LIN {X 0,Y 200.12,Z 814.334,A -85,B 0,C 180,E1 -21665.076,E2 -21665.076} C_VEL
LIN {X 0,Y 196.746,Z 821.173,A -85,B 0,C 180,E1 -21668.43,E2 -21668.43} C_VEL
LIN {X 0,Y 193.868,Z 826.716,A -85,B 0,C 180,E1 -21672.053,E2 -21672.053} C_VEL
LIN {X 0,Y 192.13,Z 830.236,A -85,B 0,C 180,E1 -21675.164,E2 -21675.164} C_VEL
LIN {X 0,Y 190.908,Z 833.5,A -85,B 0,C 180,E1 -21679.394,E2 -21679.394} C_VEL
LIN {X 0,Y 190.669,Z 835.111,A -85,B 0,C 180,E1 -21683.651,E2 -21683.651} C_VEL
LIN {X 0,Y 190.811,Z 835.331,A -85,B 0,C 180,E1 -21685.776,E2 -21685.776} C_VEL
LIN {X 0,Y 191.054,Z 835.155,A -85,B 0,C 180,E1 -21687.892,E2 -21687.892} C_VEL
LIN {X 0,Y 191.378,Z 834.552,A -85,B 0,C 180,E1 -21690,E2 -21690} C_VEL
LIN {X 0,Y 191.229,Z 834.099,A -85,B 0,C 180,E1 -21691.316,E2 -21691.316} C_VEL
LIN {X 0,Y 190.842,Z 834.419,A -85,B 0,C 180,E1 -21694.224,E2 -21694.224} C_VEL
LIN {X 0,Y 190.669,Z 834.183,A -85,B 0,C 180,E1 -21696.349,E2 -21696.349} C_VEL
LIN {X 0,Y 190.908,Z 832.465,A -85,B 0,C 180,E1 -21700.607,E2 -21700.607} C_VEL
LIN {X 0,Y 191.406,Z 831.027,A -85,B 0,C 180,E1 -21702.727,E2 -21702.727} C_VEL
LIN {X 0,Y 192.699,Z 828.062,A -85,B 0,C 180,E1 -21705.874,E2 -21705.874} C_VEL
LIN {X 0,Y 194.57,Z 824.088,A -85,B 0,C 180,E1 -21708.97,E2 -21708.97} C_VEL
LIN {X 0,Y 197.251,Z 818.323,A -85,B 0,C 180,E1 -21712.357,E2 -21712.357} C_VEL
LIN {X 0,Y 200.567,Z 811.407,A -85,B 0,C 180,E1 -21715.419,E2 -21715.419} C_VEL
LIN {X 0,Y 204.393,Z 803.243,A -85,B 0,C 180,E1 -21718.215,E2 -21718.215} C_VEL
LIN {X 0,Y 208.013,Z 794.924,A -85,B 0,C 180,E1 -21720.45,E2 -21720.45} C_VEL
LIN {X 0,Y 211.981,Z 784.694,A -85,B 0,C 180,E1 -21722.598,E2 -21722.598} C_VEL
LIN {X 0,Y 215.942,Z 773.194,A -85,B 0,C 180,E1 -21724.435,E2 -21724.435} C_VEL
LIN {X 0,Y 219.213,Z 761.827,A -85,B 0,C 180,E1 -21725.809,E2 -21725.809} C_VEL
LIN {X 0,Y 222.141,Z 748.843,A -85,B 0,C 180,E1 -21726.949,E2 -21726.949} C_VEL
LIN {X 0,Y 224.167,Z 736.06,A -85,B 0,C 180,E1 -21727.741,E2 -21727.741} C_VEL
LIN {X 0,Y 225.387,Z 722.837,A -85,B 0,C 180,E1 -21728.242,E2 -21728.242} C_VEL
LIN {X 0,Y 227.028,Z 691.593,A -85,B 0,C 180,E1 -21729.201,E2 -21729.201} C_VEL
LIN {X 0,Y 225.581,Z 668.952,A -85,B 0,C 180,E1 -21730.555,E2 -21730.555} C_VEL
LIN {X 0,Y 224.9,Z 662.654,A -85,B 0,C 180,E1 -21731.012,E2 -21731.012} C_VEL
LIN {X 0,Y 219.226,Z 646.641,A -85,B 0,C 180,E1 -21733.317,E2 -21733.317} C_VEL
LIN {X 0,Y 217.376,Z 642.169,A -85,B 0,C 180,E1 -21734.081,E2 -21734.081} C_VEL
LIN {X 0,Y 210.802,Z 631.796,A -85,B 0,C 180,E1 -21736.717,E2 -21736.717} C_VEL
LIN {X 0,Y 205.693,Z 624.408,A -85,B 0,C 180,E1 -21738.968,E2 -21738.968} C_VEL
LIN {X 0,Y 202.878,Z 620.482,A -85,B 0,C 180,E1 -21740.305,E2 -21740.305} C_VEL
LIN {X 0,Y 200.044,Z 616.68,A -85,B 0,C 180,E1 -21741.734,E2 -21741.734} C_VEL
LIN {X 0,Y 197.692,Z 613.872,A -85,B 0,C 180,E1 -21742.973,E2 -21742.973} C_VEL
LIN {X 0,Y 196.534,Z 611.954,A -85,B 0,C 180,E1 -21743.647,E2 -21743.647} C_VEL
LIN {X 0,Y 194.085,Z 610.022,A -85,B 0,C 180,E1 -21744.99,E2 -21744.99} C_VEL
LIN {X 0,Y 192.896,Z 607.766,A -85,B 0,C 180,E1 -21745.774,E2 -21745.774} C_VEL
LIN {X 0,Y 192.586,Z 606.475,A -85,B 0,C 180,E1 -21746.106,E2 -21746.106} C_VEL
LIN {X 0,Y 192.657,Z 606.463,A -85,B 0,C 180,E1 -21751.691,E2 -21751.691} C_VEL
LIN {X 0,Y 192.702,Z 606.457,A -85,B 0,C 180,E1 -21756.348,E2 -21756.348} C_VEL
LIN {X 0,Y 192.778,Z 606.466,A -85,B 0,C 180,E1 -21761.414,E2 -21761.414} C_VEL
LIN {X 0,Y 192.757,Z 606.449,A -85,B 0,C 180,E1 -21765.213,E2 -21765.213} C_VEL
LIN {X 0,Y 192.941,Z 606.428,A -85,B 0,C 180,E1 -21769.566,E2 -21769.566} C_VEL
LIN {X 0,Y 192.982,Z 606.438,A -85,B 0,C 180,E1 -21773.728,E2 -21773.728} C_VEL
LIN {X 0,Y 193.259,Z 606.38,A -85,B 0,C 180,E1 -21777.916,E2 -21777.916} C_VEL
LIN {X 0,Y 193.439,Z 606.366,A -85,B 0,C 180,E1 -21780,E2 -21780} C_VEL
LIN {X 0,Y 192.973,Z 606.424,A -85,B 0,C 180,E1 -21784.177,E2 -21784.177} C_VEL
LIN {X 0,Y 193.057,Z 606.432,A -85,B 0,C 180,E1 -21788.373,E2 -21788.373} C_VEL
LIN {X 0,Y 192.805,Z 606.44,A -85,B 0,C 180,E1 -21792.633,E2 -21792.633} C_VEL
LIN {X 0,Y 192.754,Z 606.463,A -85,B 0,C 180,E1 -21796.959,E2 -21796.959} C_VEL
LIN {X 0,Y 192.7,Z 606.473,A -85,B 0,C 180,E1 -21802.8,E2 -21802.8} C_VEL
LIN {X 0,Y 192.73,Z 606.629,A -85,B 0,C 180,E1 -21803.008,E2 -21803.008} C_VEL
LIN {X 0,Y 193.555,Z 609.094,A -85,B 0,C 180,E1 -21803.628,E2 -21803.628} C_VEL
LIN {X 0,Y 195.51,Z 611.341,A -85,B 0,C 180,E1 -21804.775,E2 -21804.775} C_VEL
LIN {X 0,Y 196.99,Z 612.434,A -85,B 0,C 180,E1 -21805.561,E2 -21805.561} C_VEL
LIN {X 0,Y 198.774,Z 615.45,A -85,B 0,C 180,E1 -21806.582,E2 -21806.582} C_VEL
LIN {X 0,Y 200.997,Z 617.62,A -85,B 0,C 180,E1 -21807.693,E2 -21807.693} C_VEL
LIN {X 0,Y 203.451,Z 621.161,A -85,B 0,C 180,E1 -21808.922,E2 -21808.922} C_VEL
LIN {X 0,Y 204.958,Z 622.964,A -85,B 0,C 180,E1 -21809.621,E2 -21809.621} C_VEL
LIN {X 0,Y 208.923,Z 628.481,A -85,B 0,C 180,E1 -21811.403,E2 -21811.403} C_VEL
LIN {X 0,Y 211.895,Z 632.606,A -85,B 0,C 180,E1 -21812.651,E2 -21812.651} C_VEL
LIN {X 0,Y 216.538,Z 639.553,A -85,B 0,C 180,E1 -21814.492,E2 -21814.492} C_VEL
LIN {X 0,Y 222.348,Z 649.031,A -85,B 0,C 180,E1 -21816.633,E2 -21816.633} C_VEL
LIN {X 0,Y 228.602,Z 660.543,A -85,B 0,C 180,E1 -21818.785,E2 -21818.785} C_VEL
LIN {X 0,Y 229.105,Z 661.475,A -85,B 0,C 180,E1 -21818.949,E2 -21818.949} C_VEL
LIN {X 0,Y 227.497,Z 690.233,A -85,B 0,C 180,E1 -21819.801,E2 -21819.801} C_VEL
LIN {X 0,Y 226.656,Z 704.192,A -85,B 0,C 180,E1 -21820.346,E2 -21820.346} C_VEL
LIN {X 0,Y 225.1,Z 717.435,A -85,B 0,C 180,E1 -21821.184,E2 -21821.184} C_VEL
LIN {X 0,Y 223.055,Z 729.09,A -85,B 0,C 180,E1 -21822.233,E2 -21822.233} C_VEL
LIN {X 0,Y 220.152,Z 741.552,A -85,B 0,C 180,E1 -21823.76,E2 -21823.76} C_VEL
LIN {X 0,Y 217.15,Z 751.905,A -85,B 0,C 180,E1 -21825.4,E2 -21825.4} C_VEL
LIN {X 0,Y 213.801,Z 761.515,A -85,B 0,C 180,E1 -21827.315,E2 -21827.315} C_VEL
LIN {X 0,Y 210.529,Z 769.77,A -85,B 0,C 180,E1 -21829.387,E2 -21829.387} C_VEL
LIN {X 0,Y 206.528,Z 778.67,A -85,B 0,C 180,E1 -21832.229,E2 -21832.229} C_VEL
LIN {X 0,Y 203.016,Z 785.739,A -85,B 0,C 180,E1 -21835.167,E2 -21835.167} C_VEL
LIN {X 0,Y 199.876,Z 791.284,A -85,B 0,C 180,E1 -21838.169,E2 -21838.169} C_VEL
LIN {X 0,Y 197.26,Z 795.562,A -85,B 0,C 180,E1 -21841.251,E2 -21841.251} C_VEL
LIN {X 0,Y 195.123,Z 798.71,A -85,B 0,C 180,E1 -21844.392,E2 -21844.392} C_VEL
LIN {X 0,Y 193.95,Z 800.243,A -85,B 0,C 180,E1 -21846.51,E2 -21846.51} C_VEL
LIN {X 0,Y 193.004,Z 801.338,A -85,B 0,C 180,E1 -21848.646,E2 -21848.646} C_VEL
LIN {X 0,Y 191.694,Z 802.23,A -85,B 0,C 180,E1 -21852.945,E2 -21852.945} C_VEL
LIN {X 0,Y 191.283,Z 802.087,A -85,B 0,C 180,E1 -21855.097,E2 -21855.097} C_VEL
LIN {X 0,Y 191.049,Z 801.498,A -85,B 0,C 180,E1 -21857.249,E2 -21857.249} C_VEL
LIN {X 0,Y 191.12,Z 799.132,A -85,B 0,C 180,E1 -21861.542,E2 -21861.542} C_VEL
LIN {X 0,Y 191.571,Z 796.233,A -85,B 0,C 180,E1 -21864.738,E2 -21864.738} C_VEL
LIN {X 0,Y 192.37,Z 792.307,A -85,B 0,C 180,E1 -21867.906,E2 -21867.906} C_VEL
LIN {X 0,Y 193.447,Z 787.253,A -85,B 0,C 180,E1 -21871.041,E2 -21871.041} C_VEL
LIN {X 0,Y 194.896,Z 780.879,A -85,B 0,C 180,E1 -21874.136,E2 -21874.136} C_VEL
LIN {X 0,Y 196.846,Z 772.934,A -85,B 0,C 180,E1 -21877.178,E2 -21877.178} C_VEL
LIN {X 0,Y 198.856,Z 764.808,A -85,B 0,C 180,E1 -21879.664,E2 -21879.664} C_VEL
LIN {X 0,Y 200.966,Z 754.894,A -85,B 0,C 180,E1 -21882.112,E2 -21882.112} C_VEL
LIN {X 0,Y 203.25,Z 743.364,A -85,B 0,C 180,E1 -21884.328,E2 -21884.328} C_VEL
LIN {X 0,Y 204.991,Z 732.793,A -85,B 0,C 180,E1 -21885.918,E2 -21885.918} C_VEL
LIN {X 0,Y 206.257,Z 723.793,A -85,B 0,C 180,E1 -21886.978,E2 -21886.978} C_VEL
LIN {X 0,Y 206.049,Z 721.845,A -85,B 0,C 180,E1 -21887.246,E2 -21887.246} C_VEL
LIN {X 0,Y 205.46,Z 720.362,A -85,B 0,C 180,E1 -21887.495,E2 -21887.495} C_VEL
LIN {X 0,Y 203.842,Z 732.893,A -85,B 0,C 180,E1 -21888.988,E2 -21888.988} C_VEL
LIN {X 0,Y 201.992,Z 744.543,A -85,B 0,C 180,E1 -21890.792,E2 -21890.792} C_VEL
LIN {X 0,Y 200.128,Z 754.446,A -85,B 0,C 180,E1 -21892.723,E2 -21892.723} C_VEL
LIN {X 0,Y 198.076,Z 764.576,A -85,B 0,C 180,E1 -21895.199,E2 -21895.199} C_VEL
LIN {X 0,Y 196.25,Z 773.003,A -85,B 0,C 180,E1 -21897.745,E2 -21897.745} C_VEL
LIN {X 0,Y 194.673,Z 780.071,A -85,B 0,C 180,E1 -21900.359,E2 -21900.359} C_VEL
LIN {X 0,Y 193.143,Z 787.462,A -85,B 0,C 180,E1 -21903.782,E2 -21903.782} C_VEL
LIN {X 0,Y 192.006,Z 793.453,A -85,B 0,C 180,E1 -21907.421,E2 -21907.421} C_VEL
LIN {X 0,Y 191.316,Z 797.226,A -85,B 0,C 180,E1 -21910.425,E2 -21910.425} C_VEL
LIN {X 0,Y 190.912,Z 800.782,A -85,B 0,C 180,E1 -21914.381,E2 -21914.381} C_VEL
LIN {X 0,Y 191.154,Z 802.884,A -85,B 0,C 180,E1 -21918.563,E2 -21918.563} C_VEL
LIN {X 0,Y 191.756,Z 803.442,A -85,B 0,C 180,E1 -21921.46,E2 -21921.46} C_VEL
LIN {X 0,Y 192.666,Z 803.238,A -85,B 0,C 180,E1 -21924.293,E2 -21924.293} C_VEL
LIN {X 0,Y 193.884,Z 802.31,A -85,B 0,C 180,E1 -21927.062,E2 -21927.062} C_VEL
LIN {X 0,Y 196.291,Z 799.661,A -85,B 0,C 180,E1 -21931.095,E2 -21931.095} C_VEL
LIN {X 0,Y 198.467,Z 796.735,A -85,B 0,C 180,E1 -21933.893,E2 -21933.893} C_VEL
LIN {X 0,Y 201.004,Z 792.853,A -85,B 0,C 180,E1 -21936.673,E2 -21936.673} C_VEL
LIN {X 0,Y 204.708,Z 786.776,A -85,B 0,C 180,E1 -21939.921,E2 -21939.921} C_VEL
LIN {X 0,Y 208.621,Z 779.506,A -85,B 0,C 180,E1 -21942.856,E2 -21942.856} C_VEL
LIN {X 0,Y 212.161,Z 772.164,A -85,B 0,C 180,E1 -21945.189,E2 -21945.189} C_VEL
LIN {X 0,Y 216.012,Z 763.265,A -85,B 0,C 180,E1 -21947.43,E2 -21947.43} C_VEL
LIN {X 0,Y 219.818,Z 752.988,A -85,B 0,C 180,E1 -21949.464,E2 -21949.464} C_VEL
LIN {X 0,Y 223.238,Z 741.939,A -85,B 0,C 180,E1 -21951.172,E2 -21951.172} C_VEL
LIN {X 0,Y 226.14,Z 730.481,A -85,B 0,C 180,E1 -21952.556,E2 -21952.556} C_VEL
LIN {X 0,Y 228.608,Z 717.196,A -85,B 0,C 180,E1 -21953.765,E2 -21953.765} C_VEL
LIN {X 0,Y 230.282,Z 704.049,A -85,B 0,C 180,E1 -21954.604,E2 -21954.604} C_VEL
LIN {X 0,Y 233.633,Z 664.942,A -85,B 0,C 180,E1 -21956.045,E2 -21956.045} C_VEL
LIN {X 0,Y 233.694,Z 662.933,A -85,B 0,C 180,E1 -21956.154,E2 -21956.154} C_VEL
LIN {X 0,Y 228.771,Z 653.042,A -85,B 0,C 180,E1 -21958.575,E2 -21958.575} C_VEL
LIN {X 0,Y 223.573,Z 644.616,A -85,B 0,C 180,E1 -21961.401,E2 -21961.401} C_VEL
LIN {X 0,Y 220.882,Z 640.179,A -85,B 0,C 180,E1 -21963.094,E2 -21963.094} C_VEL
LIN {X 0,Y 219.611,Z 638.316,A -85,B 0,C 180,E1 -21963.928,E2 -21963.928} C_VEL
LIN {X 0,Y 216.914,Z 634.667,A -85,B 0,C 180,E1 -21965.899,E2 -21965.899} C_VEL
LIN {X 0,Y 214.346,Z 631.703,A -85,B 0,C 180,E1 -21967.981,E2 -21967.981} C_VEL
LIN {X 0,Y 213.334,Z 629.707,A -85,B 0,C 180,E1 -21969.036,E2 -21969.036} C_VEL
LIN {X 0,Y 210.621,Z 627.078,A -85,B 0,C 180,E1 -21971.915,E2 -21971.915} C_VEL
LIN {X 0,Y 209.368,Z 624.536,A -85,B 0,C 180,E1 -21973.862,E2 -21973.862} C_VEL
LIN {X 0,Y 207.116,Z 623.322,A -85,B 0,C 180,E1 -21978.264,E2 -21978.264} C_VEL
LIN {X 0,Y 206.61,Z 623.792,A -85,B 0,C 180,E1 -21979.887,E2 -21979.887} C_VEL
LIN {X 0,Y 206.124,Z 625.393,A -85,B 0,C 180,E1 -21981.473,E2 -21981.473} C_VEL
LIN {X 0,Y 205.668,Z 631.128,A -85,B 0,C 180,E1 -21985.656,E2 -21985.656} C_VEL
LIN {X 0,Y 205.893,Z 632.049,A -85,B 0,C 180,E1 -21986.744,E2 -21986.744} C_VEL
LIN {X 0,Y 206.917,Z 634.357,A -85,B 0,C 180,E1 -21989.521,E2 -21989.521} C_VEL
LIN {X 0,Y 209.94,Z 639.333,A -85,B 0,C 180,E1 -21994.02,E2 -21994.02} C_VEL
LIN {X 0,Y 213.894,Z 646.761,A -85,B 0,C 180,E1 -21998.085,E2 -21998.085} C_VEL
LIN {X 0,Y 217.081,Z 653.246,A -85,B 0,C 180,E1 -22000.715,E2 -22000.715} C_VEL
LIN {X 0,Y 219.756,Z 658.788,A -85,B 0,C 180,E1 -22002.587,E2 -22002.587} C_VEL
LIN {X 0,Y 223.079,Z 666.597,A -85,B 0,C 180,E1 -22004.746,E2 -22004.746} C_VEL
LIN {X 0,Y 226.39,Z 675.777,A -85,B 0,C 180,E1 -22006.747,E2 -22006.747} C_VEL
LIN {X 0,Y 226.951,Z 691.065,A -85,B 0,C 180,E1 -22008.006,E2 -22008.006} C_VEL
LIN {X 0,Y 226.935,Z 698.487,A -85,B 0,C 180,E1 -22008.49,E2 -22008.49} C_VEL
LIN {X 0,Y 224.042,Z 728.913,A -85,B 0,C 180,E1 -22009.623,E2 -22009.623} C_VEL
LIN {X 0,Y 221.659,Z 742.96,A -85,B 0,C 180,E1 -22010.436,E2 -22010.436} C_VEL
LIN {X 0,Y 218.562,Z 755.539,A -85,B 0,C 180,E1 -22011.464,E2 -22011.464} C_VEL
LIN {X 0,Y 214.895,Z 767.424,A -85,B 0,C 180,E1 -22012.77,E2 -22012.77} C_VEL
LIN {X 0,Y 210.955,Z 778.281,A -85,B 0,C 180,E1 -22014.338,E2 -22014.338} C_VEL
LIN {X 0,Y 206.292,Z 789.283,A -85,B 0,C 180,E1 -22016.386,E2 -22016.386} C_VEL
LIN {X 0,Y 201.372,Z 799.951,A -85,B 0,C 180,E1 -22019.018,E2 -22019.018} C_VEL
LIN {X 0,Y 196.911,Z 808.526,A -85,B 0,C 180,E1 -22021.777,E2 -22021.777} C_VEL
LIN {X 0,Y 192.54,Z 816.583,A -85,B 0,C 180,E1 -22025.181,E2 -22025.181} C_VEL
LIN {X 0,Y 189.62,Z 822.117,A -85,B 0,C 180,E1 -22028.246,E2 -22028.246} C_VEL
LIN {X 0,Y 187.083,Z 826.527,A -85,B 0,C 180,E1 -22031.379,E2 -22031.379} C_VEL
LIN {X 0,Y 185.253,Z 829.916,A -85,B 0,C 180,E1 -22034.6,E2 -22034.6} C_VEL
LIN {X 0,Y 184.403,Z 831.675,A -85,B 0,C 180,E1 -22036.781,E2 -22036.781} C_VEL
LIN {X 0,Y 183.605,Z 833.941,A -85,B 0,C 180,E1 -22041.193,E2 -22041.193} C_VEL
LIN {X 0,Y 183.664,Z 834.63,A -85,B 0,C 180,E1 -22044.215,E2 -22044.215} C_VEL
LIN {X 0,Y 183.971,Z 834.424,A -85,B 0,C 180,E1 -22047.811,E2 -22047.811} C_VEL
LIN {X 0,Y 184.265,Z 833.477,A -85,B 0,C 180,E1 -22050.546,E2 -22050.546} C_VEL
LIN {X 0,Y 183.642,Z 833.713,A -85,B 0,C 180,E1 -22055.717,E2 -22055.717} C_VEL
LIN {X 0,Y 183.603,Z 832.973,A -85,B 0,C 180,E1 -22058.807,E2 -22058.807} C_VEL
LIN {X 0,Y 184.427,Z 830.537,A -85,B 0,C 180,E1 -22063.217,E2 -22063.217} C_VEL
LIN {X 0,Y 185.826,Z 827.63,A -85,B 0,C 180,E1 -22066.478,E2 -22066.478} C_VEL
LIN {X 0,Y 187.843,Z 823.721,A -85,B 0,C 180,E1 -22069.677,E2 -22069.677} C_VEL
LIN {X 0,Y 190.335,Z 818.696,A -85,B 0,C 180,E1 -22072.81,E2 -22072.81} C_VEL
LIN {X 0,Y 193.544,Z 812.421,A -85,B 0,C 180,E1 -22075.832,E2 -22075.832} C_VEL
LIN {X 0,Y 197.446,Z 804.63,A -85,B 0,C 180,E1 -22078.719,E2 -22078.719} C_VEL
LIN {X 0,Y 201.92,Z 794.934,A -85,B 0,C 180,E1 -22081.472,E2 -22081.472} C_VEL
LIN {X 0,Y 206.046,Z 784.901,A -85,B 0,C 180,E1 -22083.659,E2 -22083.659} C_VEL
LIN {X 0,Y 210.153,Z 773.575,A -85,B 0,C 180,E1 -22085.524,E2 -22085.524} C_VEL
LIN {X 0,Y 213.523,Z 762.489,A -85,B 0,C 180,E1 -22086.918,E2 -22086.918} C_VEL
LIN {X 0,Y 216.544,Z 750.025,A -85,B 0,C 180,E1 -22088.071,E2 -22088.071} C_VEL
LIN {X 0,Y 218.826,Z 736.752,A -85,B 0,C 180,E1 -22088.932,E2 -22088.932} C_VEL
LIN {X 0,Y 220.048,Z 725.276,A -85,B 0,C 180,E1 -22089.416,E2 -22089.416} C_VEL
LIN {X 0,Y 221.908,Z 692.411,A -85,B 0,C 180,E1 -22090.44,E2 -22090.44} C_VEL
LIN {X 0,Y 220.639,Z 670.867,A -85,B 0,C 180,E1 -22091.767,E2 -22091.767} C_VEL
LIN {X 0,Y 220.188,Z 665.856,A -85,B 0,C 180,E1 -22092.127,E2 -22092.127} C_VEL
LIN {X 0,Y 215.242,Z 651.377,A -85,B 0,C 180,E1 -22094.268,E2 -22094.268} C_VEL
LIN {X 0,Y 213.378,Z 646.747,A -85,B 0,C 180,E1 -22095.083,E2 -22095.083} C_VEL
LIN {X 0,Y 206.373,Z 635.432,A -85,B 0,C 180,E1 -22098.08,E2 -22098.08} C_VEL
LIN {X 0,Y 200.052,Z 626.343,A -85,B 0,C 180,E1 -22101.111,E2 -22101.111} C_VEL
LIN {X 0,Y 197.181,Z 622.528,A -85,B 0,C 180,E1 -22102.624,E2 -22102.624} C_VEL
LIN {X 0,Y 194.719,Z 619.272,A -85,B 0,C 180,E1 -22104.01,E2 -22104.01} C_VEL
LIN {X 0,Y 194.026,Z 618.292,A -85,B 0,C 180,E1 -22104.422,E2 -22104.422} C_VEL
LIN {X 0,Y 191.421,Z 615.809,A -85,B 0,C 180,E1 -22105.951,E2 -22105.951} C_VEL
LIN {X 0,Y 190.049,Z 613.108,A -85,B 0,C 180,E1 -22106.915,E2 -22106.915} C_VEL
LIN {X 0,Y 187.378,Z 611.316,A -85,B 0,C 180,E1 -22108.64,E2 -22108.64} C_VEL
LIN {X 0,Y 185.921,Z 608.849,A -85,B 0,C 180,E1 -22109.786,E2 -22109.786} C_VEL
LIN {X 0,Y 185.557,Z 607.348,A -85,B 0,C 180,E1 -22110.191,E2 -22110.191} C_VEL
LIN {X 0,Y 185.585,Z 607.353,A -85,B 0,C 180,E1 -22115.382,E2 -22115.382} C_VEL
LIN {X 0,Y 185.691,Z 607.353,A -85,B 0,C 180,E1 -22121.115,E2 -22121.115} C_VEL
LIN {X 0,Y 185.692,Z 607.324,A -85,B 0,C 180,E1 -22124.637,E2 -22124.637} C_VEL
LIN {X 0,Y 185.885,Z 607.308,A -85,B 0,C 180,E1 -22129.418,E2 -22129.418} C_VEL
LIN {X 0,Y 185.945,Z 607.309,A -85,B 0,C 180,E1 -22133.489,E2 -22133.489} C_VEL
LIN {X 0,Y 186.203,Z 607.258,A -85,B 0,C 180,E1 -22137.837,E2 -22137.837} C_VEL
LIN {X 0,Y 186.402,Z 607.241,A -85,B 0,C 180,E1 -22140,E2 -22140} C_VEL
LIN {X 0,Y 185.92,Z 607.3,A -85,B 0,C 180,E1 -22144.336,E2 -22144.336} C_VEL
LIN {X 0,Y 186.004,Z 607.314,A -85,B 0,C 180,E1 -22148.693,E2 -22148.693} C_VEL
LIN {X 0,Y 185.73,Z 607.322,A -85,B 0,C 180,E1 -22153.123,E2 -22153.123} C_VEL
LIN {X 0,Y 185.686,Z 607.335,A -85,B 0,C 180,E1 -22157.625,E2 -22157.625} C_VEL
LIN {X 0,Y 185.69,Z 607.389,A -85,B 0,C 180,E1 -22158.884,E2 -22158.884} C_VEL
LIN {X 0,Y 186.351,Z 609.679,A -85,B 0,C 180,E1 -22159.522,E2 -22159.522} C_VEL
LIN {X 0,Y 187.933,Z 611.811,A -85,B 0,C 180,E1 -22160.695,E2 -22160.695} C_VEL
LIN {X 0,Y 190.258,Z 613.373,A -85,B 0,C 180,E1 -22162.177,E2 -22162.177} C_VEL
LIN {X 0,Y 192.032,Z 616.47,A -85,B 0,C 180,E1 -22163.382,E2 -22163.382} C_VEL
LIN {X 0,Y 194.504,Z 618.874,A -85,B 0,C 180,E1 -22164.814,E2 -22164.814} C_VEL
LIN {X 0,Y 196.873,Z 622.256,A -85,B 0,C 180,E1 -22166.172,E2 -22166.172} C_VEL
LIN {X 0,Y 198.553,Z 624.143,A -85,B 0,C 180,E1 -22167.054,E2 -22167.054} C_VEL
LIN {X 0,Y 201.189,Z 627.641,A -85,B 0,C 180,E1 -22168.401,E2 -22168.401} C_VEL
LIN {X 0,Y 205.7,Z 633.976,A -85,B 0,C 180,E1 -22170.543,E2 -22170.543} C_VEL
LIN {X 0,Y 210.561,Z 640.986,A -85,B 0,C 180,E1 -22172.651,E2 -22172.651} C_VEL
LIN {X 0,Y 217.786,Z 652.676,A -85,B 0,C 180,E1 -22175.511,E2 -22175.511} C_VEL
LIN {X 0,Y 223.948,Z 664.331,A -85,B 0,C 180,E1 -22177.767,E2 -22177.767} C_VEL
LIN {X 0,Y 222.381,Z 690.882,A -85,B 0,C 180,E1 -22178.56,E2 -22178.56} C_VEL
LIN {X 0,Y 221.499,Z 704.795,A -85,B 0,C 180,E1 -22179.112,E2 -22179.112} C_VEL
LIN {X 0,Y 219.943,Z 717.573,A -85,B 0,C 180,E1 -22179.926,E2 -22179.926} C_VEL
LIN {X 0,Y 217.734,Z 729.689,A -85,B 0,C 180,E1 -22181.02,E2 -22181.02} C_VEL
LIN {X 0,Y 214.709,Z 742.158,A -85,B 0,C 180,E1 -22182.569,E2 -22182.569} C_VEL
LIN {X 0,Y 211.621,Z 752.417,A -85,B 0,C 180,E1 -22184.22,E2 -22184.22} C_VEL
LIN {X 0,Y 208.093,Z 762.126,A -85,B 0,C 180,E1 -22186.185,E2 -22186.185} C_VEL
LIN {X 0,Y 204.302,Z 771.192,A -85,B 0,C 180,E1 -22188.533,E2 -22188.533} C_VEL
LIN {X 0,Y 200.135,Z 779.954,A -85,B 0,C 180,E1 -22191.443,E2 -22191.443} C_VEL
LIN {X 0,Y 196.45,Z 786.852,A -85,B 0,C 180,E1 -22194.456,E2 -22194.456} C_VEL
LIN {X 0,Y 193.692,Z 791.498,A -85,B 0,C 180,E1 -22197.026,E2 -22197.026} C_VEL
LIN {X 0,Y 190.872,Z 795.87,A -85,B 0,C 180,E1 -22200.194,E2 -22200.194} C_VEL
LIN {X 0,Y 188.581,Z 799.104,A -85,B 0,C 180,E1 -22203.436,E2 -22203.436} C_VEL
LIN {X 0,Y 187.287,Z 800.679,A -85,B 0,C 180,E1 -22205.621,E2 -22205.621} C_VEL
LIN {X 0,Y 186.229,Z 801.838,A -85,B 0,C 180,E1 -22207.829,E2 -22207.829} C_VEL
LIN {X 0,Y 184.87,Z 802.806,A -85,B 0,C 180,E1 -22211.879,E2 -22211.879} C_VEL
LIN {X 0,Y 184.295,Z 802.726,A -85,B 0,C 180,E1 -22214.518,E2 -22214.518} C_VEL
LIN {X 0,Y 184.003,Z 802.211,A -85,B 0,C 180,E1 -22216.752,E2 -22216.752} C_VEL
LIN {X 0,Y 183.917,Z 801.263,A -85,B 0,C 180,E1 -22218.985,E2 -22218.985} C_VEL
LIN {X 0,Y 184.174,Z 798.684,A -85,B 0,C 180,E1 -22222.817,E2 -22222.817} C_VEL
LIN {X 0,Y 184.954,Z 794.679,A -85,B 0,C 180,E1 -22226.733,E2 -22226.733} C_VEL
LIN {X 0,Y 185.89,Z 790.106,A -85,B 0,C 180,E1 -22230,E2 -22230} C_VEL
LIN {X 0,Y 187.555,Z 783.198,A -85,B 0,C 180,E1 -22233.76,E2 -22233.76} C_VEL
LIN {X 0,Y 189.466,Z 775.71,A -85,B 0,C 180,E1 -22236.924,E2 -22236.924} C_VEL
LIN {X 0,Y 191.872,Z 766.274,A -85,B 0,C 180,E1 -22240.019,E2 -22240.019} C_VEL
LIN {X 0,Y 194.054,Z 756.597,A -85,B 0,C 180,E1 -22242.55,E2 -22242.55} C_VEL
LIN {X 0,Y 196.251,Z 745.958,A -85,B 0,C 180,E1 -22244.73,E2 -22244.73} C_VEL
LIN {X 0,Y 198.227,Z 735.059,A -85,B 0,C 180,E1 -22246.477,E2 -22246.477} C_VEL
LIN {X 0,Y 198.855,Z 730.991,A -85,B 0,C 180,E1 -22247.026,E2 -22247.026} C_VEL
LIN {X 0,Y 198.717,Z 729.466,A -85,B 0,C 180,E1 -22247.272,E2 -22247.272} C_VEL
LIN {X 0,Y 197.908,Z 728.01,A -85,B 0,C 180,E1 -22247.638,E2 -22247.638} C_VEL
LIN {X 0,Y 196.084,Z 739.963,A -85,B 0,C 180,E1 -22249.339,E2 -22249.339} C_VEL
LIN {X 0,Y 194.193,Z 750.33,A -85,B 0,C 180,E1 -22251.217,E2 -22251.217} C_VEL
LIN {X 0,Y 191.921,Z 761.382,A -85,B 0,C 180,E1 -22253.753,E2 -22253.753} C_VEL
LIN {X 0,Y 190.008,Z 770.415,A -85,B 0,C 180,E1 -22256.349,E2 -22256.349} C_VEL
LIN {X 0,Y 188.229,Z 778.044,A -85,B 0,C 180,E1 -22259.037,E2 -22259.037} C_VEL
LIN {X 0,Y 186.644,Z 785.381,A -85,B 0,C 180,E1 -22262.27,E2 -22262.27} C_VEL
LIN {X 0,Y 185.317,Z 791.717,A -85,B 0,C 180,E1 -22265.831,E2 -22265.831} C_VEL
LIN {X 0,Y 184.519,Z 795.928,A -85,B 0,C 180,E1 -22268.865,E2 -22268.865} C_VEL
LIN {X 0,Y 184.005,Z 799.206,A -85,B 0,C 180,E1 -22271.918,E2 -22271.918} C_VEL
LIN {X 0,Y 183.824,Z 801.637,A -85,B 0,C 180,E1 -22274.994,E2 -22274.994} C_VEL
LIN {X 0,Y 183.876,Z 802.557,A -85,B 0,C 180,E1 -22276.568,E2 -22276.568} C_VEL
LIN {X 0,Y 184.274,Z 803.743,A -85,B 0,C 180,E1 -22279.708,E2 -22279.708} C_VEL
LIN {X 0,Y 185.093,Z 804.108,A -85,B 0,C 180,E1 -22282.878,E2 -22282.878} C_VEL
LIN {X 0,Y 186.299,Z 803.629,A -85,B 0,C 180,E1 -22286.09,E2 -22286.09} C_VEL
LIN {X 0,Y 187.985,Z 802.249,A -85,B 0,C 180,E1 -22289.3,E2 -22289.3} C_VEL
LIN {X 0,Y 190.144,Z 799.892,A -85,B 0,C 180,E1 -22292.505,E2 -22292.505} C_VEL
LIN {X 0,Y 193.57,Z 795.443,A -85,B 0,C 180,E1 -22296.46,E2 -22296.46} C_VEL
LIN {X 0,Y 197.044,Z 790.349,A -85,B 0,C 180,E1 -22299.65,E2 -22299.65} C_VEL
LIN {X 0,Y 201.205,Z 783.448,A -85,B 0,C 180,E1 -22302.856,E2 -22302.856} C_VEL
LIN {X 0,Y 205.735,Z 774.988,A -85,B 0,C 180,E1 -22305.838,E2 -22305.838} C_VEL
LIN {X 0,Y 210.248,Z 765.258,A -85,B 0,C 180,E1 -22308.43,E2 -22308.43} C_VEL
LIN {X 0,Y 214.364,Z 755.033,A -85,B 0,C 180,E1 -22310.565,E2 -22310.565} C_VEL
LIN {X 0,Y 218.133,Z 743.833,A -85,B 0,C 180,E1 -22312.363,E2 -22312.363} C_VEL
LIN {X 0,Y 221.141,Z 732.709,A -85,B 0,C 180,E1 -22313.763,E2 -22313.763} C_VEL
LIN {X 0,Y 223.738,Z 720.218,A -85,B 0,C 180,E1 -22314.965,E2 -22314.965} C_VEL
LIN {X 0,Y 225.631,Z 706.998,A -85,B 0,C 180,E1 -22315.86,E2 -22315.86} C_VEL
LIN {X 0,Y 226.873,Z 693.522,A -85,B 0,C 180,E1 -22316.448,E2 -22316.448} C_VEL
LIN {X 0,Y 229.279,Z 666.002,A -85,B 0,C 180,E1 -22317.466,E2 -22317.466} C_VEL
LIN {X 0,Y 225.266,Z 657.892,A -85,B 0,C 180,E1 -22319.607,E2 -22319.607} C_VEL
LIN {X 0,Y 219.546,Z 647.958,A -85,B 0,C 180,E1 -22323.07,E2 -22323.07} C_VEL
LIN {X 0,Y 217.391,Z 644.633,A -85,B 0,C 180,E1 -22324.567,E2 -22324.567} C_VEL
LIN {X 0,Y 214.932,Z 641.187,A -85,B 0,C 180,E1 -22326.445,E2 -22326.445} C_VEL
LIN {X 0,Y 212.336,Z 637.932,A -85,B 0,C 180,E1 -22328.724,E2 -22328.724} C_VEL
LIN {X 0,Y 211.388,Z 636.283,A -85,B 0,C 180,E1 -22329.733,E2 -22329.733} C_VEL
LIN {X 0,Y 208.839,Z 633.391,A -85,B 0,C 180,E1 -22332.759,E2 -22332.759} C_VEL
LIN {X 0,Y 208.043,Z 631.579,A -85,B 0,C 180,E1 -22334.108,E2 -22334.108} C_VEL
LIN {X 0,Y 205.821,Z 630.198,A -85,B 0,C 180,E1 -22338.928,E2 -22338.928} C_VEL
LIN {X 0,Y 205.344,Z 630.045,A -85,B 0,C 180,E1 -22342.472,E2 -22342.472} C_VEL
LIN {X 0,Y 205.893,Z 632.049,A -85,B 0,C 180,E1 -22346.744,E2 -22346.744} C_VEL
LIN {X 0,Y 206.343,Z 633.802,A -85,B 0,C 180,E1 -22348.3,E2 -22348.3} C_VEL
LIN {X 0,Y 206.733,Z 636.637,A -85,B 0,C 180,E1 -22349.742,E2 -22349.742} C_VEL
LIN {X 0,Y 208.228,Z 645.71,A -85,B 0,C 180,E1 -22353.384,E2 -22353.384} C_VEL
LIN {X 0,Y 208.929,Z 647.563,A -85,B 0,C 180,E1 -22354.345,E2 -22354.345} C_VEL
LIN {X 0,Y 211.745,Z 653.027,A -85,B 0,C 180,E1 -22357.361,E2 -22357.361} C_VEL
LIN {X 0,Y 214.546,Z 658.958,A -85,B 0,C 180,E1 -22359.818,E2 -22359.818} C_VEL
LIN {X 0,Y 217.054,Z 664.588,A -85,B 0,C 180,E1 -22361.751,E2 -22361.751} C_VEL
LIN {X 0,Y 220.304,Z 672.852,A -85,B 0,C 180,E1 -22364.045,E2 -22364.045} C_VEL
LIN {X 0,Y 222.479,Z 679.187,A -85,B 0,C 180,E1 -22365.457,E2 -22365.457} C_VEL
LIN {X 0,Y 222.816,Z 693.204,A -85,B 0,C 180,E1 -22366.63,E2 -22366.63} C_VEL
LIN {X 0,Y 222.731,Z 699.438,A -85,B 0,C 180,E1 -22367.049,E2 -22367.049} C_VEL
LIN {X 0,Y 219.813,Z 728.15,A -85,B 0,C 180,E1 -22368.129,E2 -22368.129} C_VEL
LIN {X 0,Y 217.459,Z 741.643,A -85,B 0,C 180,E1 -22368.904,E2 -22368.904} C_VEL
LIN {X 0,Y 214.278,Z 754.376,A -85,B 0,C 180,E1 -22369.935,E2 -22369.935} C_VEL
LIN {X 0,Y 210.441,Z 766.361,A -85,B 0,C 180,E1 -22371.232,E2 -22371.232} C_VEL
LIN {X 0,Y 206.288,Z 777.296,A -85,B 0,C 180,E1 -22372.792,E2 -22372.792} C_VEL
LIN {X 0,Y 201.419,Z 788.293,A -85,B 0,C 180,E1 -22374.851,E2 -22374.851} C_VEL
LIN {X 0,Y 197.002,Z 797.31,A -85,B 0,C 180,E1 -22377.042,E2 -22377.042} C_VEL
LIN {X 0,Y 192.178,Z 806.28,A -85,B 0,C 180,E1 -22379.813,E2 -22379.813} C_VEL
LIN {X 0,Y 187.965,Z 813.592,A -85,B 0,C 180,E1 -22382.741,E2 -22382.741} C_VEL
LIN {X 0,Y 184.345,Z 819.736,A -85,B 0,C 180,E1 -22385.95,E2 -22385.95} C_VEL
LIN {X 0,Y 181.19,Z 824.995,A -85,B 0,C 180,E1 -22389.569,E2 -22389.569} C_VEL
LIN {X 0,Y 178.983,Z 828.595,A -85,B 0,C 180,E1 -22392.873,E2 -22392.873} C_VEL
LIN {X 0,Y 177.443,Z 831.253,A -85,B 0,C 180,E1 -22396.253,E2 -22396.253} C_VEL
LIN {X 0,Y 176.554,Z 833.387,A -85,B 0,C 180,E1 -22400.838,E2 -22400.838} C_VEL
LIN {X 0,Y 176.597,Z 833.975,A -85,B 0,C 180,E1 -22404.224,E2 -22404.224} C_VEL
LIN {X 0,Y 176.893,Z 833.656,A -85,B 0,C 180,E1 -22407.723,E2 -22407.723} C_VEL
LIN {X 0,Y 177.204,Z 832.597,A -85,B 0,C 180,E1 -22410.71,E2 -22410.71} C_VEL
LIN {X 0,Y 176.583,Z 833.145,A -85,B 0,C 180,E1 -22415.731,E2 -22415.731} C_VEL
LIN {X 0,Y 176.552,Z 832.431,A -85,B 0,C 180,E1 -22419.162,E2 -22419.162} C_VEL
LIN {X 0,Y 177.468,Z 830.051,A -85,B 0,C 180,E1 -22423.745,E2 -22423.745} C_VEL
LIN {X 0,Y 178.982,Z 827.204,A -85,B 0,C 180,E1 -22427.127,E2 -22427.127} C_VEL
LIN {X 0,Y 181.143,Z 823.358,A -85,B 0,C 180,E1 -22430.437,E2 -22430.437} C_VEL
LIN {X 0,Y 183.772,Z 818.4,A -85,B 0,C 180,E1 -22433.673,E2 -22433.673} C_VEL
LIN {X 0,Y 187.17,Z 812.2,A -85,B 0,C 180,E1 -22436.781,E2 -22436.781} C_VEL
LIN {X 0,Y 191.251,Z 804.535,A -85,B 0,C 180,E1 -22439.741,E2 -22439.741} C_VEL
LIN {X 0,Y 195.896,Z 794.944,A -85,B 0,C 180,E1 -22442.556,E2 -22442.556} C_VEL
LIN {X 0,Y 200.191,Z 785.076,A -85,B 0,C 180,E1 -22444.783,E2 -22444.783} C_VEL
LIN {X 0,Y 204.442,Z 773.957,A -85,B 0,C 180,E1 -22446.675,E2 -22446.675} C_VEL
LIN {X 0,Y 207.918,Z 763.111,A -85,B 0,C 180,E1 -22448.088,E2 -22448.088} C_VEL
LIN {X 0,Y 211.032,Z 751.157,A -85,B 0,C 180,E1 -22449.253,E2 -22449.253} C_VEL
LIN {X 0,Y 213.431,Z 738.328,A -85,B 0,C 180,E1 -22450.142,E2 -22450.142} C_VEL
LIN {X 0,Y 214.903,Z 726.041,A -85,B 0,C 180,E1 -22450.701,E2 -22450.701} C_VEL
LIN {X 0,Y 216.906,Z 693.325,A -85,B 0,C 180,E1 -22451.734,E2 -22451.734} C_VEL
LIN {X 0,Y 215.674,Z 670.666,A -85,B 0,C 180,E1 -22453.18,E2 -22453.18} C_VEL
LIN {X 0,Y 215.153,Z 667.514,A -85,B 0,C 180,E1 -22453.489,E2 -22453.489} C_VEL
LIN {X 0,Y 209.88,Z 652.035,A -85,B 0,C 180,E1 -22455.939,E2 -22455.939} C_VEL
LIN {X 0,Y 203.142,Z 640.902,A -85,B 0,C 180,E1 -22458.976,E2 -22458.976} C_VEL
LIN {X 0,Y 196.985,Z 631.86,A -85,B 0,C 180,E1 -22462.091,E2 -22462.091} C_VEL
LIN {X 0,Y 194.275,Z 628.252,A -85,B 0,C 180,E1 -22463.594,E2 -22463.594} C_VEL
LIN {X 0,Y 191.533,Z 624.508,A -85,B 0,C 180,E1 -22465.237,E2 -22465.237} C_VEL
LIN {X 0,Y 188.846,Z 621.602,A -85,B 0,C 180,E1 -22466.921,E2 -22466.921} C_VEL
LIN {X 0,Y 187.696,Z 619.579,A -85,B 0,C 180,E1 -22467.753,E2 -22467.753} C_VEL
LIN {X 0,Y 185.016,Z 617.293,A -85,B 0,C 180,E1 -22469.623,E2 -22469.623} C_VEL
LIN {X 0,Y 183.486,Z 614.453,A -85,B 0,C 180,E1 -22470.923,E2 -22470.923} C_VEL
LIN {X 0,Y 183.321,Z 614.074,A -85,B 0,C 180,E1 -22471.075,E2 -22471.075} C_VEL
LIN {X 0,Y 180.626,Z 612.438,A -85,B 0,C 180,E1 -22473.265,E2 -22473.265} C_VEL
LIN {X 0,Y 179.151,Z 610.365,A -85,B 0,C 180,E1 -22474.724,E2 -22474.724} C_VEL
LIN {X 0,Y 178.536,Z 608.228,A -85,B 0,C 180,E1 -22475.54,E2 -22475.54} C_VEL
LIN {X 0,Y 178.667,Z 608.218,A -85,B 0,C 180,E1 -22481.658,E2 -22481.658} C_VEL
LIN {X 0,Y 178.653,Z 608.217,A -85,B 0,C 180,E1 -22486.347,E2 -22486.347} C_VEL
LIN {X 0,Y 178.907,Z 608.166,A -85,B 0,C 180,E1 -22490.96,E2 -22490.96} C_VEL
LIN {X 0,Y 178.865,Z 608.199,A -85,B 0,C 180,E1 -22495.493,E2 -22495.493} C_VEL
LIN {X 0,Y 179.366,Z 608.117,A -85,B 0,C 180,E1 -22500,E2 -22500} C_VEL
LIN {X 0,Y 178.868,Z 608.176,A -85,B 0,C 180,E1 -22504.507,E2 -22504.507} C_VEL
LIN {X 0,Y 178.955,Z 608.194,A -85,B 0,C 180,E1 -22509.038,E2 -22509.038} C_VEL
LIN {X 0,Y 178.691,Z 608.277,A -85,B 0,C 180,E1 -22513.577,E2 -22513.577} C_VEL
LIN {X 0,Y 179.265,Z 610.362,A -85,B 0,C 180,E1 -22514.328,E2 -22514.328} C_VEL
LIN {X 0,Y 181.206,Z 612.833,A -85,B 0,C 180,E1 -22516.186,E2 -22516.186} C_VEL
LIN {X 0,Y 183.535,Z 614.316,A -85,B 0,C 180,E1 -22518.051,E2 -22518.051} C_VEL
LIN {X 0,Y 184.982,Z 617.147,A -85,B 0,C 180,E1 -22519.293,E2 -22519.293} C_VEL
LIN {X 0,Y 187.467,Z 619.421,A -85,B 0,C 180,E1 -22521.047,E2 -22521.047} C_VEL
LIN {X 0,Y 188.102,Z 620.07,A -85,B 0,C 180,E1 -22521.478,E2 -22521.478} C_VEL
LIN {X 0,Y 190.43,Z 623.49,A -85,B 0,C 180,E1 -22523.06,E2 -22523.06} C_VEL
LIN {X 0,Y 192.137,Z 625.249,A -85,B 0,C 180,E1 -22524.087,E2 -22524.087} C_VEL
LIN {X 0,Y 194.801,Z 628.841,A -85,B 0,C 180,E1 -22525.654,E2 -22525.654} C_VEL
LIN {X 0,Y 196.167,Z 630.662,A -85,B 0,C 180,E1 -22526.414,E2 -22526.414} C_VEL
LIN {X 0,Y 199.505,Z 635.219,A -85,B 0,C 180,E1 -22528.174,E2 -22528.174} C_VEL
LIN {X 0,Y 204.921,Z 642.917,A -85,B 0,C 180,E1 -22530.768,E2 -22530.768} C_VEL
LIN {X 0,Y 211.19,Z 652.845,A -85,B 0,C 180,E1 -22533.488,E2 -22533.488} C_VEL
LIN {X 0,Y 217.281,Z 663.782,A -85,B 0,C 180,E1 -22535.904,E2 -22535.904} C_VEL
LIN {X 0,Y 218.87,Z 666.882,A -85,B 0,C 180,E1 -22536.505,E2 -22536.505} C_VEL
LIN {X 0,Y 217.394,Z 691.143,A -85,B 0,C 180,E1 -22537.243,E2 -22537.243} C_VEL
LIN {X 0,Y 216.44,Z 705.609,A -85,B 0,C 180,E1 -22537.828,E2 -22537.828} C_VEL
LIN {X 0,Y 214.799,Z 718.383,A -85,B 0,C 180,E1 -22538.654,E2 -22538.654} C_VEL
LIN {X 0,Y 212.505,Z 730.388,A -85,B 0,C 180,E1 -22539.755,E2 -22539.755} C_VEL
LIN {X 0,Y 209.363,Z 742.788,A -85,B 0,C 180,E1 -22541.316,E2 -22541.316} C_VEL
LIN {X 0,Y 206.186,Z 752.944,A -85,B 0,C 180,E1 -22542.978,E2 -22542.978} C_VEL
LIN {X 0,Y 202.46,Z 762.744,A -85,B 0,C 180,E1 -22544.988,E2 -22544.988} C_VEL
LIN {X 0,Y 198.841,Z 770.994,A -85,B 0,C 180,E1 -22547.127,E2 -22547.127} C_VEL
LIN {X 0,Y 194.445,Z 779.893,A -85,B 0,C 180,E1 -22550.094,E2 -22550.094} C_VEL
LIN {X 0,Y 190.562,Z 786.962,A -85,B 0,C 180,E1 -22553.181,E2 -22553.181} C_VEL
LIN {X 0,Y 187.581,Z 791.695,A -85,B 0,C 180,E1 -22555.807,E2 -22555.807} C_VEL
LIN {X 0,Y 184.577,Z 796.177,A -85,B 0,C 180,E1 -22559.068,E2 -22559.068} C_VEL
LIN {X 0,Y 181.839,Z 799.758,A -85,B 0,C 180,E1 -22562.741,E2 -22562.741} C_VEL
LIN {X 0,Y 179.493,Z 802.317,A -85,B 0,C 180,E1 -22566.95,E2 -22566.95} C_VEL
LIN {X 0,Y 178.544,Z 803.096,A -85,B 0,C 180,E1 -22569.252,E2 -22569.252} C_VEL
LIN {X 0,Y 177.861,Z 803.421,A -85,B 0,C 180,E1 -22571.573,E2 -22571.573} C_VEL
LIN {X 0,Y 177.338,Z 803.359,A -85,B 0,C 180,E1 -22573.894,E2 -22573.894} C_VEL
LIN {X 0,Y 176.97,Z 802.911,A -85,B 0,C 180,E1 -22576.215,E2 -22576.215} C_VEL
LIN {X 0,Y 176.837,Z 802.014,A -85,B 0,C 180,E1 -22578.539,E2 -22578.539} C_VEL
LIN {X 0,Y 177.087,Z 799.277,A -85,B 0,C 180,E1 -22582.827,E2 -22582.827} C_VEL
LIN {X 0,Y 177.824,Z 795.604,A -85,B 0,C 180,E1 -22586.601,E2 -22586.601} C_VEL
LIN {X 0,Y 178.787,Z 791.134,A -85,B 0,C 180,E1 -22590,E2 -22590} C_VEL
LIN {X 0,Y 180.489,Z 784.336,A -85,B 0,C 180,E1 -22593.907,E2 -22593.907} C_VEL
LIN {X 0,Y 182.44,Z 776.974,A -85,B 0,C 180,E1 -22597.192,E2 -22597.192} C_VEL
LIN {X 0,Y 184.45,Z 769.445,A -85,B 0,C 180,E1 -22599.873,E2 -22599.873} C_VEL
LIN {X 0,Y 186.939,Z 759.249,A -85,B 0,C 180,E1 -22602.76,E2 -22602.76} C_VEL
LIN {X 0,Y 189.235,Z 748.911,A -85,B 0,C 180,E1 -22605.068,E2 -22605.068} C_VEL
LIN {X 0,Y 191.474,Z 737.313,A -85,B 0,C 180,E1 -22607.075,E2 -22607.075} C_VEL
LIN {X 0,Y 191.387,Z 736.088,A -85,B 0,C 180,E1 -22607.3,E2 -22607.3} C_VEL
LIN {X 0,Y 190.335,Z 734.531,A -85,B 0,C 180,E1 -22607.767,E2 -22607.767} C_VEL
LIN {X 0,Y 188.407,Z 745.703,A -85,B 0,C 180,E1 -22609.616,E2 -22609.616} C_VEL
LIN {X 0,Y 186.357,Z 755.861,A -85,B 0,C 180,E1 -22611.736,E2 -22611.736} C_VEL
LIN {X 0,Y 184.222,Z 765.737,A -85,B 0,C 180,E1 -22614.317,E2 -22614.317} C_VEL
LIN {X 0,Y 182.074,Z 775.183,A -85,B 0,C 180,E1 -22617.403,E2 -22617.403} C_VEL
LIN {X 0,Y 180.112,Z 783.473,A -85,B 0,C 180,E1 -22620.857,E2 -22620.857} C_VEL
LIN {X 0,Y 178.706,Z 790.012,A -85,B 0,C 180,E1 -22624.323,E2 -22624.323} C_VEL
LIN {X 0,Y 177.683,Z 795.024,A -85,B 0,C 180,E1 -22627.714,E2 -22627.714} C_VEL
LIN {X 0,Y 177.025,Z 798.802,A -85,B 0,C 180,E1 -22631.034,E2 -22631.034} C_VEL
LIN {X 0,Y 176.768,Z 802.475,A -85,B 0,C 180,E1 -22635.695,E2 -22635.695} C_VEL
LIN {X 0,Y 177.067,Z 804.022,A -85,B 0,C 180,E1 -22638.948,E2 -22638.948} C_VEL
LIN {X 0,Y 177.793,Z 804.743,A -85,B 0,C 180,E1 -22642.238,E2 -22642.238} C_VEL
LIN {X 0,Y 179.502,Z 804.334,A -85,B 0,C 180,E1 -22646.76,E2 -22646.76} C_VEL
LIN {X 0,Y 181.068,Z 803.223,A -85,B 0,C 180,E1 -22649.696,E2 -22649.696} C_VEL
LIN {X 0,Y 184.098,Z 800.194,A -85,B 0,C 180,E1 -22653.959,E2 -22653.959} C_VEL
LIN {X 0,Y 187.896,Z 795.561,A -85,B 0,C 180,E1 -22658.035,E2 -22658.035} C_VEL
LIN {X 0,Y 191.774,Z 790.145,A -85,B 0,C 180,E1 -22661.344,E2 -22661.344} C_VEL
LIN {X 0,Y 195.57,Z 784.193,A -85,B 0,C 180,E1 -22664.121,E2 -22664.121} C_VEL
LIN {X 0,Y 199.753,Z 776.936,A -85,B 0,C 180,E1 -22666.781,E2 -22666.781} C_VEL
LIN {X 0,Y 204.327,Z 767.951,A -85,B 0,C 180,E1 -22669.346,E2 -22669.346} C_VEL
LIN {X 0,Y 208.636,Z 758.003,A -85,B 0,C 180,E1 -22671.542,E2 -22671.542} C_VEL
LIN {X 0,Y 212.307,Z 748.15,A -85,B 0,C 180,E1 -22673.248,E2 -22673.248} C_VEL
LIN {X 0,Y 215.702,Z 737.046,A -85,B 0,C 180,E1 -22674.777,E2 -22674.777} C_VEL
LIN {X 0,Y 218.746,Z 724.441,A -85,B 0,C 180,E1 -22676.087,E2 -22676.087} C_VEL
LIN {X 0,Y 220.993,Z 711.147,A -85,B 0,C 180,E1 -22677.118,E2 -22677.118} C_VEL
LIN {X 0,Y 222.396,Z 698.16,A -85,B 0,C 180,E1 -22677.766,E2 -22677.766} C_VEL
LIN {X 0,Y 225.063,Z 669.246,A -85,B 0,C 180,E1 -22678.842,E2 -22678.842} C_VEL
LIN {X 0,Y 221.754,Z 662.406,A -85,B 0,C 180,E1 -22680.762,E2 -22680.762} C_VEL
LIN {X 0,Y 216.329,Z 652.721,A -85,B 0,C 180,E1 -22684.366,E2 -22684.366} C_VEL
LIN {X 0,Y 213.226,Z 647.947,A -85,B 0,C 180,E1 -22686.802,E2 -22686.802} C_VEL
LIN {X 0,Y 210.581,Z 644.581,A -85,B 0,C 180,E1 -22689.24,E2 -22689.24} C_VEL
LIN {X 0,Y 209.768,Z 643.041,A -85,B 0,C 180,E1 -22690.154,E2 -22690.154} C_VEL
LIN {X 0,Y 207.244,Z 639.93,A -85,B 0,C 180,E1 -22693.381,E2 -22693.381} C_VEL
LIN {X 0,Y 206.576,Z 638.384,A -85,B 0,C 180,E1 -22694.597,E2 -22694.597} C_VEL
LIN {X 0,Y 204.466,Z 637.026,A -85,B 0,C 180,E1 -22700.104,E2 -22700.104} C_VEL
LIN {X 0,Y 204.225,Z 637.221,A -85,B 0,C 180,E1 -22702.821,E2 -22702.821} C_VEL
LIN {X 0,Y 204.79,Z 639.211,A -85,B 0,C 180,E1 -22706.843,E2 -22706.843} C_VEL
LIN {X 0,Y 206.781,Z 643.443,A -85,B 0,C 180,E1 -22711.336,E2 -22711.336} C_VEL
LIN {X 0,Y 208.268,Z 646.083,A -85,B 0,C 180,E1 -22713.51,E2 -22713.51} C_VEL
LIN {X 0,Y 208.929,Z 647.563,A -85,B 0,C 180,E1 -22714.345,E2 -22714.345} C_VEL
LIN {X 0,Y 209.999,Z 650.626,A -85,B 0,C 180,E1 -22715.69,E2 -22715.69} C_VEL
LIN {X 0,Y 210.857,Z 654.595,A -85,B 0,C 180,E1 -22716.87,E2 -22716.87} C_VEL
LIN {X 0,Y 213.12,Z 666.448,A -85,B 0,C 180,E1 -22719.738,E2 -22719.738} C_VEL
LIN {X 0,Y 213.965,Z 669.093,A -85,B 0,C 180,E1 -22720.518,E2 -22720.518} C_VEL
LIN {X 0,Y 217.324,Z 678.185,A -85,B 0,C 180,E1 -22723.093,E2 -22723.093} C_VEL
LIN {X 0,Y 218.736,Z 682.916,A -85,B 0,C 180,E1 -22724.162,E2 -22724.162} C_VEL
LIN {X 0,Y 218.871,Z 694.364,A -85,B 0,C 180,E1 -22725.126,E2 -22725.126} C_VEL
LIN {X 0,Y 218.693,Z 700.981,A -85,B 0,C 180,E1 -22725.561,E2 -22725.561} C_VEL
LIN {X 0,Y 215.877,Z 727.385,A -85,B 0,C 180,E1 -22726.557,E2 -22726.557} C_VEL
LIN {X 0,Y 213.32,Z 741.28,A -85,B 0,C 180,E1 -22727.357,E2 -22727.357} C_VEL
LIN {X 0,Y 210.118,Z 753.428,A -85,B 0,C 180,E1 -22728.336,E2 -22728.336} C_VEL
LIN {X 0,Y 206.133,Z 765.38,A -85,B 0,C 180,E1 -22729.626,E2 -22729.626} C_VEL
LIN {X 0,Y 201.774,Z 776.314,A -85,B 0,C 180,E1 -22731.175,E2 -22731.175} C_VEL
LIN {X 0,Y 196.703,Z 787.376,A -85,B 0,C 180,E1 -22733.241,E2 -22733.241} C_VEL
LIN {X 0,Y 192.031,Z 796.436,A -85,B 0,C 180,E1 -22735.441,E2 -22735.441} C_VEL
LIN {X 0,Y 186.909,Z 805.403,A -85,B 0,C 180,E1 -22738.237,E2 -22738.237} C_VEL
LIN {X 0,Y 182.377,Z 812.712,A -85,B 0,C 180,E1 -22741.205,E2 -22741.205} C_VEL
LIN {X 0,Y 178.554,Z 818.681,A -85,B 0,C 180,E1 -22744.345,E2 -22744.345} C_VEL
LIN {X 0,Y 175.472,Z 823.506,A -85,B 0,C 180,E1 -22747.636,E2 -22747.636} C_VEL
LIN {X 0,Y 172.842,Z 827.286,A -85,B 0,C 180,E1 -22751.017,E2 -22751.017} C_VEL
LIN {X 0,Y 170.505,Z 830.821,A -85,B 0,C 180,E1 -22755.682,E2 -22755.682} C_VEL
LIN {X 0,Y 169.499,Z 832.838,A -85,B 0,C 180,E1 -22760.453,E2 -22760.453} C_VEL
LIN {X 0,Y 169.536,Z 833.316,A -85,B 0,C 180,E1 -22764.214,E2 -22764.214} C_VEL
LIN {X 0,Y 169.817,Z 832.878,A -85,B 0,C 180,E1 -22767.628,E2 -22767.628} C_VEL
LIN {X 0,Y 170.159,Z 831.845,A -85,B 0,C 180,E1 -22770.592,E2 -22770.592} C_VEL
LIN {X 0,Y 169.62,Z 832.562,A -85,B 0,C 180,E1 -22774.753,E2 -22774.753} C_VEL
LIN {X 0,Y 169.499,Z 831.88,A -85,B 0,C 180,E1 -22779.547,E2 -22779.547} C_VEL
LIN {X 0,Y 170.529,Z 829.566,A -85,B 0,C 180,E1 -22784.316,E2 -22784.316} C_VEL
LIN {X 0,Y 172.165,Z 826.778,A -85,B 0,C 180,E1 -22787.828,E2 -22787.828} C_VEL
LIN {X 0,Y 175.068,Z 821.944,A -85,B 0,C 180,E1 -22792.07,E2 -22792.07} C_VEL
LIN {X 0,Y 178.34,Z 816.223,A -85,B 0,C 180,E1 -22795.688,E2 -22795.688} C_VEL
LIN {X 0,Y 182.218,Z 809.631,A -85,B 0,C 180,E1 -22798.823,E2 -22798.823} C_VEL
LIN {X 0,Y 186.665,Z 801.489,A -85,B 0,C 180,E1 -22801.809,E2 -22801.809} C_VEL
LIN {X 0,Y 190.856,Z 793.197,A -85,B 0,C 180,E1 -22804.163,E2 -22804.163} C_VEL
LIN {X 0,Y 194.93,Z 784.162,A -85,B 0,C 180,E1 -22806.183,E2 -22806.183} C_VEL
LIN {X 0,Y 198.812,Z 774.368,A -85,B 0,C 180,E1 -22807.893,E2 -22807.893} C_VEL
LIN {X 0,Y 202.9,Z 762.036,A -85,B 0,C 180,E1 -22809.528,E2 -22809.528} C_VEL
LIN {X 0,Y 206.125,Z 750.066,A -85,B 0,C 180,E1 -22810.679,E2 -22810.679} C_VEL
LIN {X 0,Y 208.526,Z 737.531,A -85,B 0,C 180,E1 -22811.542,E2 -22811.542} C_VEL
LIN {X 0,Y 210.129,Z 724.472,A -85,B 0,C 180,E1 -22812.123,E2 -22812.123} C_VEL
LIN {X 0,Y 212.024,Z 694.396,A -85,B 0,C 180,E1 -22813.082,E2 -22813.082} C_VEL
LIN {X 0,Y 210.928,Z 671.897,A -85,B 0,C 180,E1 -22814.558,E2 -22814.558} C_VEL
LIN {X 0,Y 207.046,Z 659.53,A -85,B 0,C 180,E1 -22816.494,E2 -22816.494} C_VEL
LIN {X 0,Y 205.584,Z 655.887,A -85,B 0,C 180,E1 -22817.209,E2 -22817.209} C_VEL
LIN {X 0,Y 199.796,Z 646.177,A -85,B 0,C 180,E1 -22819.98,E2 -22819.98} C_VEL
LIN {X 0,Y 194.359,Z 637.865,A -85,B 0,C 180,E1 -22822.889,E2 -22822.889} C_VEL
LIN {X 0,Y 191.285,Z 633.737,A -85,B 0,C 180,E1 -22824.683,E2 -22824.683} C_VEL
LIN {X 0,Y 189.035,Z 630.646,A -85,B 0,C 180,E1 -22826.105,E2 -22826.105} C_VEL
LIN {X 0,Y 186.282,Z 627.301,A -85,B 0,C 180,E1 -22827.957,E2 -22827.957} C_VEL
LIN {X 0,Y 185.388,Z 625.941,A -85,B 0,C 180,E1 -22828.623,E2 -22828.623} C_VEL
LIN {X 0,Y 182.762,Z 623.299,A -85,B 0,C 180,E1 -22830.591,E2 -22830.591} C_VEL
LIN {X 0,Y 181.224,Z 620.69,A -85,B 0,C 180,E1 -22831.951,E2 -22831.951} C_VEL
LIN {X 0,Y 178.639,Z 618.705,A -85,B 0,C 180,E1 -22834.22,E2 -22834.22} C_VEL
LIN {X 0,Y 177.135,Z 616.201,A -85,B 0,C 180,E1 -22835.857,E2 -22835.857} C_VEL
LIN {X 0,Y 176.763,Z 615.108,A -85,B 0,C 180,E1 -22836.346,E2 -22836.346} C_VEL
LIN {X 0,Y 173.992,Z 613.64,A -85,B 0,C 180,E1 -22839.549,E2 -22839.549} C_VEL
LIN {X 0,Y 171.951,Z 610.68,A -85,B 0,C 180,E1 -22842.916,E2 -22842.916} C_VEL
LIN {X 0,Y 171.593,Z 609.078,A -85,B 0,C 180,E1 -22843.951,E2 -22843.951} C_VEL
LIN {X 0,Y 171.844,Z 609.046,A -85,B 0,C 180,E1 -22850.585,E2 -22850.585} C_VEL
LIN {X 0,Y 171.814,Z 609.079,A -85,B 0,C 180,E1 -22855.307,E2 -22855.307} C_VEL
LIN {X 0,Y 172.329,Z 608.992,A -85,B 0,C 180,E1 -22860,E2 -22860} C_VEL
LIN {X 0,Y 171.842,Z 609.237,A -85,B 0,C 180,E1 -22865.574,E2 -22865.574} C_VEL
LIN {X 0,Y 172.92,Z 612.005,A -85,B 0,C 180,E1 -22867.737,E2 -22867.737} C_VEL
LIN {X 0,Y 175.53,Z 614.49,A -85,B 0,C 180,E1 -22871.27,E2 -22871.27} C_VEL
LIN {X 0,Y 176.908,Z 615.25,A -85,B 0,C 180,E1 -22872.767,E2 -22872.767} C_VEL
LIN {X 0,Y 178.201,Z 617.957,A -85,B 0,C 180,E1 -22874.27,E2 -22874.27} C_VEL
LIN {X 0,Y 180.496,Z 620.218,A -85,B 0,C 180,E1 -22876.397,E2 -22876.397} C_VEL
LIN {X 0,Y 181.597,Z 621.042,A -85,B 0,C 180,E1 -22877.308,E2 -22877.308} C_VEL
LIN {X 0,Y 183.647,Z 624.342,A -85,B 0,C 180,E1 -22879.056,E2 -22879.056} C_VEL
LIN {X 0,Y 185.942,Z 626.489,A -85,B 0,C 180,E1 -22880.714,E2 -22880.714} C_VEL
LIN {X 0,Y 188.446,Z 630.026,A -85,B 0,C 180,E1 -22882.474,E2 -22882.474} C_VEL
LIN {X 0,Y 189.862,Z 631.656,A -85,B 0,C 180,E1 -22883.376,E2 -22883.376} C_VEL
LIN {X 0,Y 193.571,Z 636.697,A -85,B 0,C 180,E1 -22885.613,E2 -22885.613} C_VEL
LIN {X 0,Y 198.913,Z 644.178,A -85,B 0,C 180,E1 -22888.489,E2 -22888.489} C_VEL
LIN {X 0,Y 205.37,Z 654.18,A -85,B 0,C 180,E1 -22891.572,E2 -22891.572} C_VEL
LIN {X 0,Y 211.229,Z 664.487,A -85,B 0,C 180,E1 -22894.107,E2 -22894.107} C_VEL
LIN {X 0,Y 213.894,Z 669.632,A -85,B 0,C 180,E1 -22895.191,E2 -22895.191} C_VEL
LIN {X 0,Y 212.131,Z 698.588,A -85,B 0,C 180,E1 -22896.115,E2 -22896.115} C_VEL
LIN {X 0,Y 210.846,Z 711.909,A -85,B 0,C 180,E1 -22896.801,E2 -22896.801} C_VEL
LIN {X 0,Y 208.803,Z 724.408,A -85,B 0,C 180,E1 -22897.762,E2 -22897.762} C_VEL
LIN {X 0,Y 206.011,Z 736.745,A -85,B 0,C 180,E1 -22899.096,E2 -22899.096} C_VEL
LIN {X 0,Y 202.449,Z 748.826,A -85,B 0,C 180,E1 -22900.847,E2 -22900.847} C_VEL
LIN {X 0,Y 198.685,Z 759.143,A -85,B 0,C 180,E1 -22902.78,E2 -22902.78} C_VEL
LIN {X 0,Y 194.362,Z 769.025,A -85,B 0,C 180,E1 -22905.163,E2 -22905.163} C_VEL
LIN {X 0,Y 190.62,Z 776.637,A -85,B 0,C 180,E1 -22907.509,E2 -22907.509} C_VEL
LIN {X 0,Y 186.747,Z 783.655,A -85,B 0,C 180,E1 -22910.226,E2 -22910.226} C_VEL
LIN {X 0,Y 182.693,Z 790.251,A -85,B 0,C 180,E1 -22913.535,E2 -22913.535} C_VEL
LIN {X 0,Y 179.342,Z 795.061,A -85,B 0,C 180,E1 -22916.728,E2 -22916.728} C_VEL
LIN {X 0,Y 176.452,Z 798.846,A -85,B 0,C 180,E1 -22920.142,E2 -22920.142} C_VEL
LIN {X 0,Y 174.096,Z 801.552,A -85,B 0,C 180,E1 -22923.638,E2 -22923.638} C_VEL
LIN {X 0,Y 172.798,Z 802.794,A -85,B 0,C 180,E1 -22926.002,E2 -22926.002} C_VEL
LIN {X 0,Y 171.753,Z 803.632,A -85,B 0,C 180,E1 -22928.391,E2 -22928.391} C_VEL
LIN {X 0,Y 170.905,Z 804.028,A -85,B 0,C 180,E1 -22931.052,E2 -22931.052} C_VEL
LIN {X 0,Y 169.953,Z 803.585,A -85,B 0,C 180,E1 -22935.634,E2 -22935.634} C_VEL
LIN {X 0,Y 169.784,Z 802.763,A -85,B 0,C 180,E1 -22938.056,E2 -22938.056} C_VEL
LIN {X 0,Y 170.005,Z 799.881,A -85,B 0,C 180,E1 -22942.822,E2 -22942.822} C_VEL
LIN {X 0,Y 170.698,Z 796.511,A -85,B 0,C 180,E1 -22946.459,E2 -22946.459} C_VEL
LIN {X 0,Y 171.677,Z 792.131,A -85,B 0,C 180,E1 -22950,E2 -22950} C_VEL
LIN {X 0,Y 173.428,Z 785.474,A -85,B 0,C 180,E1 -22954.067,E2 -22954.067} C_VEL
LIN {X 0,Y 175.395,Z 778.229,A -85,B 0,C 180,E1 -22957.482,E2 -22957.482} C_VEL
LIN {X 0,Y 177.476,Z 770.827,A -85,B 0,C 180,E1 -22960.265,E2 -22960.265} C_VEL
LIN {X 0,Y 179.85,Z 761.879,A -85,B 0,C 180,E1 -22962.984,E2 -22962.984} C_VEL
LIN {X 0,Y 182.139,Z 751.985,A -85,B 0,C 180,E1 -22965.383,E2 -22965.383} C_VEL
LIN {X 0,Y 183.989,Z 743.499,A -85,B 0,C 180,E1 -22967.042,E2 -22967.042} C_VEL
LIN {X 0,Y 184.048,Z 742.053,A -85,B 0,C 180,E1 -22967.322,E2 -22967.322} C_VEL
LIN {X 0,Y 182.747,Z 740.326,A -85,B 0,C 180,E1 -22967.88,E2 -22967.88} C_VEL
LIN {X 0,Y 180.419,Z 752.24,A -85,B 0,C 180,E1 -22970.203,E2 -22970.203} C_VEL
LIN {X 0,Y 177.994,Z 763.26,A -85,B 0,C 180,E1 -22972.948,E2 -22972.948} C_VEL
LIN {X 0,Y 176.048,Z 771.663,A -85,B 0,C 180,E1 -22975.562,E2 -22975.562} C_VEL
LIN {X 0,Y 174.279,Z 778.838,A -85,B 0,C 180,E1 -22978.276,E2 -22978.276} C_VEL
LIN {X 0,Y 172.763,Z 785.425,A -85,B 0,C 180,E1 -22981.319,E2 -22981.319} C_VEL
LIN {X 0,Y 171.321,Z 791.877,A -85,B 0,C 180,E1 -22985.051,E2 -22985.051} C_VEL
LIN {X 0,Y 170.403,Z 796.418,A -85,B 0,C 180,E1 -22988.406,E2 -22988.406} C_VEL
LIN {X 0,Y 169.834,Z 800.017,A -85,B 0,C 180,E1 -22991.852,E2 -22991.852} C_VEL
LIN {X 0,Y 169.681,Z 802.609,A -85,B 0,C 180,E1 -22995.241,E2 -22995.241} C_VEL
LIN {X 0,Y 169.935,Z 804.321,A -85,B 0,C 180,E1 -22998.569,E2 -22998.569} C_VEL
LIN {X 0,Y 170.599,Z 805.247,A -85,B 0,C 180,E1 -23001.834,E2 -23001.834} C_VEL
LIN {X 0,Y 171.645,Z 805.442,A -85,B 0,C 180,E1 -23005.024,E2 -23005.024} C_VEL
LIN {X 0,Y 173.203,Z 804.803,A -85,B 0,C 180,E1 -23008.44,E2 -23008.44} C_VEL
LIN {X 0,Y 175.312,Z 803.252,A -85,B 0,C 180,E1 -23011.875,E2 -23011.875} C_VEL
LIN {X 0,Y 177.977,Z 800.73,A -85,B 0,C 180,E1 -23015.259,E2 -23015.259} C_VEL
LIN {X 0,Y 181.17,Z 797.133,A -85,B 0,C 180,E1 -23018.59,E2 -23018.59} C_VEL
LIN {X 0,Y 185.658,Z 791.418,A -85,B 0,C 180,E1 -23022.372,E2 -23022.372} C_VEL
LIN {X 0,Y 190.193,Z 784.815,A -85,B 0,C 180,E1 -23025.556,E2 -23025.556} C_VEL
LIN {X 0,Y 195.076,Z 776.757,A -85,B 0,C 180,E1 -23028.513,E2 -23028.513} C_VEL
LIN {X 0,Y 199.861,Z 767.654,A -85,B 0,C 180,E1 -23031.051,E2 -23031.051} C_VEL
LIN {X 0,Y 204.72,Z 756.892,A -85,B 0,C 180,E1 -23033.38,E2 -23033.38} C_VEL
LIN {X 0,Y 208.834,Z 746.043,A -85,B 0,C 180,E1 -23035.174,E2 -23035.174} C_VEL
LIN {X 0,Y 212.446,Z 734.1,A -85,B 0,C 180,E1 -23036.706,E2 -23036.706} C_VEL
LIN {X 0,Y 215.273,Z 721.898,A -85,B 0,C 180,E1 -23037.899,E2 -23037.899} C_VEL
LIN {X 0,Y 217.407,Z 708.653,A -85,B 0,C 180,E1 -23038.814,E2 -23038.814} C_VEL
LIN {X 0,Y 218.732,Z 696.017,A -85,B 0,C 180,E1 -23039.382,E2 -23039.382} C_VEL
LIN {X 0,Y 220.948,Z 672.468,A -85,B 0,C 180,E1 -23040.296,E2 -23040.296} C_VEL
LIN {X 0,Y 218.483,Z 667.261,A -85,B 0,C 180,E1 -23041.887,E2 -23041.887} C_VEL
LIN {X 0,Y 213.59,Z 658.062,A -85,B 0,C 180,E1 -23045.452,E2 -23045.452} C_VEL
LIN {X 0,Y 210.968,Z 654.179,A -85,B 0,C 180,E1 -23047.658,E2 -23047.658} C_VEL
LIN {X 0,Y 208.381,Z 650.258,A -85,B 0,C 180,E1 -23050.313,E2 -23050.313} C_VEL
LIN {X 0,Y 205.528,Z 646.115,A -85,B 0,C 180,E1 -23054.284,E2 -23054.284} C_VEL
LIN {X 0,Y 205.207,Z 645.264,A -85,B 0,C 180,E1 -23054.997,E2 -23054.997} C_VEL
LIN {X 0,Y 203.316,Z 644.031,A -85,B 0,C 180,E1 -23060.223,E2 -23060.223} C_VEL
LIN {X 0,Y 203.093,Z 644.322,A -85,B 0,C 180,E1 -23062.955,E2 -23062.955} C_VEL
LIN {X 0,Y 203.689,Z 646.429,A -85,B 0,C 180,E1 -23067,E2 -23067} C_VEL
LIN {X 0,Y 206.156,Z 651.659,A -85,B 0,C 180,E1 -23072.205,E2 -23072.205} C_VEL
LIN {X 0,Y 209.557,Z 658.918,A -85,B 0,C 180,E1 -23076.469,E2 -23076.469} C_VEL
LIN {X 0,Y 212.144,Z 664.814,A -85,B 0,C 180,E1 -23078.957,E2 -23078.957} C_VEL
LIN {X 0,Y 213.965,Z 669.093,A -85,B 0,C 180,E1 -23080.518,E2 -23080.518} C_VEL
LIN {X 0,Y 214.767,Z 671.856,A -85,B 0,C 180,E1 -23081.23,E2 -23081.23} C_VEL
LIN {X 0,Y 215.441,Z 676.883,A -85,B 0,C 180,E1 -23082.043,E2 -23082.043} C_VEL
LIN {X 0,Y 215.587,Z 682.453,A -85,B 0,C 180,E1 -23082.617,E2 -23082.617} C_VEL
LIN {X 0,Y 215.105,Z 698.485,A -85,B 0,C 180,E1 -23083.784,E2 -23083.784} C_VEL
LIN {X 0,Y 214.692,Z 704.18,A -85,B 0,C 180,E1 -23084.076,E2 -23084.076} C_VEL
LIN {X 0,Y 212.006,Z 727.334,A -85,B 0,C 180,E1 -23084.963,E2 -23084.963} C_VEL
LIN {X 0,Y 209.478,Z 740.441,A -85,B 0,C 180,E1 -23085.714,E2 -23085.714} C_VEL
LIN {X 0,Y 206.143,Z 752.636,A -85,B 0,C 180,E1 -23086.678,E2 -23086.678} C_VEL
LIN {X 0,Y 202.029,Z 764.599,A -85,B 0,C 180,E1 -23087.961,E2 -23087.961} C_VEL
LIN {X 0,Y 197.464,Z 775.548,A -85,B 0,C 180,E1 -23089.494,E2 -23089.494} C_VEL
LIN {X 0,Y 192.151,Z 786.556,A -85,B 0,C 180,E1 -23091.555,E2 -23091.555} C_VEL
LIN {X 0,Y 187.175,Z 795.587,A -85,B 0,C 180,E1 -23093.746,E2 -23093.746} C_VEL
LIN {X 0,Y 181.798,Z 804.567,A -85,B 0,C 180,E1 -23096.574,E2 -23096.574} C_VEL
LIN {X 0,Y 176.935,Z 811.911,A -85,B 0,C 180,E1 -23099.574,E2 -23099.574} C_VEL
LIN {X 0,Y 172.168,Z 818.731,A -85,B 0,C 180,E1 -23103.319,E2 -23103.319} C_VEL
LIN {X 0,Y 168.882,Z 823.371,A -85,B 0,C 180,E1 -23106.713,E2 -23106.713} C_VEL
LIN {X 0,Y 166.099,Z 827.018,A -85,B 0,C 180,E1 -23110.215,E2 -23110.215} C_VEL
LIN {X 0,Y 163.588,Z 830.41,A -85,B 0,C 180,E1 -23115.063,E2 -23115.063} C_VEL
LIN {X 0,Y 162.884,Z 831.538,A -85,B 0,C 180,E1 -23117.542,E2 -23117.542} C_VEL
LIN {X 0,Y 162.352,Z 832.593,A -85,B 0,C 180,E1 -23122.538,E2 -23122.538} C_VEL
LIN {X 0,Y 162.55,Z 832.549,A -85,B 0,C 180,E1 -23125.039,E2 -23125.039} C_VEL
LIN {X 0,Y 162.742,Z 832.096,A -85,B 0,C 180,E1 -23127.525,E2 -23127.525} C_VEL
LIN {X 0,Y 163.119,Z 831.13,A -85,B 0,C 180,E1 -23130.463,E2 -23130.463} C_VEL
LIN {X 0,Y 162.518,Z 831.94,A -85,B 0,C 180,E1 -23134.962,E2 -23134.962} C_VEL
LIN {X 0,Y 162.471,Z 831.316,A -85,B 0,C 180,E1 -23139.964,E2 -23139.964} C_VEL
LIN {X 0,Y 162.894,Z 830.409,A -85,B 0,C 180,E1 -23142.458,E2 -23142.458} C_VEL
LIN {X 0,Y 164.723,Z 827.368,A -85,B 0,C 180,E1 -23147.377,E2 -23147.377} C_VEL
LIN {X 0,Y 166.923,Z 823.984,A -85,B 0,C 180,E1 -23150.969,E2 -23150.969} C_VEL
LIN {X 0,Y 169.733,Z 819.548,A -85,B 0,C 180,E1 -23154.46,E2 -23154.46} C_VEL
LIN {X 0,Y 173.223,Z 813.939,A -85,B 0,C 180,E1 -23157.812,E2 -23157.812} C_VEL
LIN {X 0,Y 177.497,Z 806.99,A -85,B 0,C 180,E1 -23160.979,E2 -23160.979} C_VEL
LIN {X 0,Y 182.367,Z 798.321,A -85,B 0,C 180,E1 -23163.972,E2 -23163.972} C_VEL
LIN {X 0,Y 186.794,Z 789.469,A -85,B 0,C 180,E1 -23166.339,E2 -23166.339} C_VEL
LIN {X 0,Y 191.183,Z 779.77,A -85,B 0,C 180,E1 -23168.339,E2 -23168.339} C_VEL
LIN {X 0,Y 195.382,Z 769.112,A -85,B 0,C 180,E1 -23170.013,E2 -23170.013} C_VEL
LIN {X 0,Y 199.198,Z 757.211,A -85,B 0,C 180,E1 -23171.415,E2 -23171.415} C_VEL
LIN {X 0,Y 202.221,Z 744.887,A -85,B 0,C 180,E1 -23172.494,E2 -23172.494} C_VEL
LIN {X 0,Y 204.426,Z 731.97,A -85,B 0,C 180,E1 -23173.268,E2 -23173.268} C_VEL
LIN {X 0,Y 205.822,Z 717.16,A -85,B 0,C 180,E1 -23173.816,E2 -23173.816} C_VEL
LIN {X 0,Y 207.222,Z 694.903,A -85,B 0,C 180,E1 -23174.536,E2 -23174.536} C_VEL
LIN {X 0,Y 206.37,Z 674.688,A -85,B 0,C 180,E1 -23175.897,E2 -23175.897} C_VEL
LIN {X 0,Y 204.695,Z 668.711,A -85,B 0,C 180,E1 -23176.805,E2 -23176.805} C_VEL
LIN {X 0,Y 202.048,Z 660.914,A -85,B 0,C 180,E1 -23178.215,E2 -23178.215} C_VEL
LIN {X 0,Y 196.834,Z 651.901,A -85,B 0,C 180,E1 -23180.851,E2 -23180.851} C_VEL
LIN {X 0,Y 191.29,Z 643.174,A -85,B 0,C 180,E1 -23183.996,E2 -23183.996} C_VEL
LIN {X 0,Y 186.704,Z 636.872,A -85,B 0,C 180,E1 -23186.919,E2 -23186.919} C_VEL
LIN {X 0,Y 183.812,Z 633.032,A -85,B 0,C 180,E1 -23189.004,E2 -23189.004} C_VEL
LIN {X 0,Y 180.328,Z 628.897,A -85,B 0,C 180,E1 -23191.8,E2 -23191.8} C_VEL
LIN {X 0,Y 179.477,Z 627.357,A -85,B 0,C 180,E1 -23192.606,E2 -23192.606} C_VEL
LIN {X 0,Y 176.79,Z 625.035,A -85,B 0,C 180,E1 -23195.112,E2 -23195.112} C_VEL
LIN {X 0,Y 174.976,Z 621.885,A -85,B 0,C 180,E1 -23197.253,E2 -23197.253} C_VEL
LIN {X 0,Y 172.304,Z 620.079,A -85,B 0,C 180,E1 -23200.646,E2 -23200.646} C_VEL
LIN {X 0,Y 170.526,Z 616.855,A -85,B 0,C 180,E1 -23204.001,E2 -23204.001} C_VEL
LIN {X 0,Y 170.364,Z 616.217,A -85,B 0,C 180,E1 -23204.446,E2 -23204.446} C_VEL
LIN {X 0,Y 167.932,Z 614.96,A -85,B 0,C 180,E1 -23212.787,E2 -23212.787} C_VEL
LIN {X 0,Y 168.668,Z 615.094,A -85,B 0,C 180,E1 -23220.121,E2 -23220.121} C_VEL
LIN {X 0,Y 170.623,Z 616.284,A -85,B 0,C 180,E1 -23225.021,E2 -23225.021} C_VEL
LIN {X 0,Y 171.923,Z 619.18,A -85,B 0,C 180,E1 -23227.635,E2 -23227.635} C_VEL
LIN {X 0,Y 174.613,Z 621.581,A -85,B 0,C 180,E1 -23231.283,E2 -23231.283} C_VEL
LIN {X 0,Y 175.367,Z 622.227,A -85,B 0,C 180,E1 -23232.146,E2 -23232.146} C_VEL
LIN {X 0,Y 177.1,Z 625.232,A -85,B 0,C 180,E1 -23234.141,E2 -23234.141} C_VEL
LIN {X 0,Y 179.76,Z 627.663,A -85,B 0,C 180,E1 -23236.594,E2 -23236.594} C_VEL
LIN {X 0,Y 181.989,Z 631.082,A -85,B 0,C 180,E1 -23238.553,E2 -23238.553} C_VEL
LIN {X 0,Y 183.924,Z 633.027,A -85,B 0,C 180,E1 -23240.016,E2 -23240.016} C_VEL
LIN {X 0,Y 186.695,Z 636.782,A -85,B 0,C 180,E1 -23242.017,E2 -23242.017} C_VEL
LIN {X 0,Y 191.088,Z 642.848,A -85,B 0,C 180,E1 -23244.835,E2 -23244.835} C_VEL
LIN {X 0,Y 196.244,Z 650.356,A -85,B 0,C 180,E1 -23247.747,E2 -23247.747} C_VEL
LIN {X 0,Y 202.035,Z 659.549,A -85,B 0,C 180,E1 -23250.653,E2 -23250.653} C_VEL
LIN {X 0,Y 207.476,Z 669.364,A -85,B 0,C 180,E1 -23253.137,E2 -23253.137} C_VEL
LIN {X 0,Y 209.022,Z 672.447,A -85,B 0,C 180,E1 -23253.812,E2 -23253.812} C_VEL
LIN {X 0,Y 207.11,Z 702.628,A -85,B 0,C 180,E1 -23254.846,E2 -23254.846} C_VEL
LIN {X 0,Y 205.546,Z 715.76,A -85,B 0,C 180,E1 -23255.594,E2 -23255.594} C_VEL
LIN {X 0,Y 203.175,Z 728.331,A -85,B 0,C 180,E1 -23256.674,E2 -23256.674} C_VEL
LIN {X 0,Y 200.494,Z 739.146,A -85,B 0,C 180,E1 -23257.938,E2 -23257.938} C_VEL
LIN {X 0,Y 197.162,Z 749.74,A -85,B 0,C 180,E1 -23259.519,E2 -23259.519} C_VEL
LIN {X 0,Y 193.323,Z 759.775,A -85,B 0,C 180,E1 -23261.429,E2 -23261.429} C_VEL
LIN {X 0,Y 189.253,Z 768.766,A -85,B 0,C 180,E1 -23263.604,E2 -23263.604} C_VEL
LIN {X 0,Y 184.864,Z 777.296,A -85,B 0,C 180,E1 -23266.247,E2 -23266.247} C_VEL
LIN {X 0,Y 180.46,Z 784.89,A -85,B 0,C 180,E1 -23269.284,E2 -23269.284} C_VEL
LIN {X 0,Y 177.006,Z 790.204,A -85,B 0,C 180,E1 -23272.018,E2 -23272.018} C_VEL
LIN {X 0,Y 173.265,Z 795.326,A -85,B 0,C 180,E1 -23275.399,E2 -23275.399} C_VEL
LIN {X 0,Y 170.151,Z 799.204,A -85,B 0,C 180,E1 -23278.916,E2 -23278.916} C_VEL
LIN {X 0,Y 167.592,Z 801.992,A -85,B 0,C 180,E1 -23282.531,E2 -23282.531} C_VEL
LIN {X 0,Y 166.155,Z 803.274,A -85,B 0,C 180,E1 -23284.978,E2 -23284.978} C_VEL
LIN {X 0,Y 164.993,Z 804.151,A -85,B 0,C 180,E1 -23287.459,E2 -23287.459} C_VEL
LIN {X 0,Y 163.946,Z 804.638,A -85,B 0,C 180,E1 -23290.578,E2 -23290.578} C_VEL
LIN {X 0,Y 162.952,Z 804.258,A -85,B 0,C 180,E1 -23295.003,E2 -23295.003} C_VEL
LIN {X 0,Y 162.718,Z 803.497,A -85,B 0,C 180,E1 -23297.529,E2 -23297.529} C_VEL
LIN {X 0,Y 162.695,Z 802.29,A -85,B 0,C 180,E1 -23300.05,E2 -23300.05} C_VEL
LIN {X 0,Y 162.923,Z 800.482,A -85,B 0,C 180,E1 -23302.818,E2 -23302.818} C_VEL
LIN {X 0,Y 163.557,Z 797.42,A -85,B 0,C 180,E1 -23306.305,E2 -23306.305} C_VEL
LIN {X 0,Y 164.561,Z 793.125,A -85,B 0,C 180,E1 -23310,E2 -23310} C_VEL
LIN {X 0,Y 166.066,Z 787.644,A -85,B 0,C 180,E1 -23313.64,E2 -23313.64} C_VEL
LIN {X 0,Y 167.977,Z 780.809,A -85,B 0,C 180,E1 -23317.21,E2 -23317.21} C_VEL
LIN {X 0,Y 170.504,Z 772.206,A -85,B 0,C 180,E1 -23320.689,E2 -23320.689} C_VEL
LIN {X 0,Y 172.985,Z 763.404,A -85,B 0,C 180,E1 -23323.509,E2 -23323.509} C_VEL
LIN {X 0,Y 175.362,Z 753.777,A -85,B 0,C 180,E1 -23325.993,E2 -23325.993} C_VEL
LIN {X 0,Y 176.723,Z 747.37,A -85,B 0,C 180,E1 -23327.361,E2 -23327.361} C_VEL
LIN {X 0,Y 175.132,Z 745.6,A -85,B 0,C 180,E1 -23328.044,E2 -23328.044} C_VEL
LIN {X 0,Y 172.665,Z 757.023,A -85,B 0,C 180,E1 -23330.581,E2 -23330.581} C_VEL
LIN {X 0,Y 170.115,Z 767.933,A -85,B 0,C 180,E1 -23333.678,E2 -23333.678} C_VEL
LIN {X 0,Y 168.01,Z 776.471,A -85,B 0,C 180,E1 -23336.723,E2 -23336.723} C_VEL
LIN {X 0,Y 165.921,Z 784.913,A -85,B 0,C 180,E1 -23340.549,E2 -23340.549} C_VEL
LIN {X 0,Y 164.323,Z 791.911,A -85,B 0,C 180,E1 -23344.62,E2 -23344.62} C_VEL
LIN {X 0,Y 163.379,Z 796.495,A -85,B 0,C 180,E1 -23348.053,E2 -23348.053} C_VEL
LIN {X 0,Y 162.779,Z 800.105,A -85,B 0,C 180,E1 -23351.521,E2 -23351.521} C_VEL
LIN {X 0,Y 162.622,Z 803.605,A -85,B 0,C 180,E1 -23356.253,E2 -23356.253} C_VEL
LIN {X 0,Y 163.245,Z 805.519,A -85,B 0,C 180,E1 -23360.797,E2 -23360.797} C_VEL
LIN {X 0,Y 164.267,Z 806.108,A -85,B 0,C 180,E1 -23364.378,E2 -23364.378} C_VEL
LIN {X 0,Y 165.807,Z 805.854,A -85,B 0,C 180,E1 -23367.964,E2 -23367.964} C_VEL
LIN {X 0,Y 168.706,Z 804.077,A -85,B 0,C 180,E1 -23372.726,E2 -23372.726} C_VEL
LIN {X 0,Y 171.144,Z 802.046,A -85,B 0,C 180,E1 -23375.754,E2 -23375.754} C_VEL
LIN {X 0,Y 173.898,Z 799.325,A -85,B 0,C 180,E1 -23378.67,E2 -23378.67} C_VEL
LIN {X 0,Y 177.515,Z 795.287,A -85,B 0,C 180,E1 -23381.834,E2 -23381.834} C_VEL
LIN {X 0,Y 181.843,Z 789.805,A -85,B 0,C 180,E1 -23385.059,E2 -23385.059} C_VEL
LIN {X 0,Y 186.713,Z 782.819,A -85,B 0,C 180,E1 -23388.134,E2 -23388.134} C_VEL
LIN {X 0,Y 191.68,Z 774.821,A -85,B 0,C 180,E1 -23390.841,E2 -23390.841} C_VEL
LIN {X 0,Y 196.713,Z 765.377,A -85,B 0,C 180,E1 -23393.333,E2 -23393.333} C_VEL
LIN {X 0,Y 201.593,Z 754.538,A -85,B 0,C 180,E1 -23395.501,E2 -23395.501} C_VEL
LIN {X 0,Y 205.851,Z 743.138,A -85,B 0,C 180,E1 -23397.261,E2 -23397.261} C_VEL
LIN {X 0,Y 209.701,Z 729.918,A -85,B 0,C 180,E1 -23398.792,E2 -23398.792} C_VEL
LIN {X 0,Y 212.389,Z 717.402,A -85,B 0,C 180,E1 -23399.887,E2 -23399.887} C_VEL
LIN {X 0,Y 214.233,Z 704.418,A -85,B 0,C 180,E1 -23400.668,E2 -23400.668} C_VEL
LIN {X 0,Y 217.132,Z 675.825,A -85,B 0,C 180,E1 -23401.792,E2 -23401.792} C_VEL
LIN {X 0,Y 212.891,Z 667.344,A -85,B 0,C 180,E1 -23404.895,E2 -23404.895} C_VEL
LIN {X 0,Y 210.877,Z 663.45,A -85,B 0,C 180,E1 -23406.594,E2 -23406.594} C_VEL
LIN {X 0,Y 209.031,Z 660.633,A -85,B 0,C 180,E1 -23408.309,E2 -23408.309} C_VEL
LIN {X 0,Y 206.311,Z 656.256,A -85,B 0,C 180,E1 -23411.372,E2 -23411.372} C_VEL
LIN {X 0,Y 204.145,Z 652.986,A -85,B 0,C 180,E1 -23414.677,E2 -23414.677} C_VEL
LIN {X 0,Y 203.93,Z 652.294,A -85,B 0,C 180,E1 -23415.218,E2 -23415.218} C_VEL
LIN {X 0,Y 202.362,Z 651.185,A -85,B 0,C 180,E1 -23419.264,E2 -23419.264} C_VEL
LIN {X 0,Y 201.957,Z 651.199,A -85,B 0,C 180,E1 -23422.507,E2 -23422.507} C_VEL
LIN {X 0,Y 202.438,Z 653.302,A -85,B 0,C 180,E1 -23426.662,E2 -23426.662} C_VEL
LIN {X 0,Y 204.762,Z 658.578,A -85,B 0,C 180,E1 -23431.903,E2 -23431.903} C_VEL
LIN {X 0,Y 207.621,Z 665.37,A -85,B 0,C 180,E1 -23435.783,E2 -23435.783} C_VEL
LIN {X 0,Y 209.94,Z 671.094,A -85,B 0,C 180,E1 -23438.231,E2 -23438.231} C_VEL
LIN {X 0,Y 212.046,Z 676.566,A -85,B 0,C 180,E1 -23440.153,E2 -23440.153} C_VEL
LIN {X 0,Y 214.709,Z 684.536,A -85,B 0,C 180,E1 -23442.364,E2 -23442.364} C_VEL
LIN {X 0,Y 215.176,Z 686.443,A -85,B 0,C 180,E1 -23442.768,E2 -23442.768} C_VEL
LIN {X 0,Y 215.105,Z 698.485,A -85,B 0,C 180,E1 -23443.784,E2 -23443.784} C_VEL
LIN {X 0,Y 214.864,Z 702.302,A -85,B 0,C 180,E1 -23443.985,E2 -23443.985} C_VEL
LIN {X 0,Y 213.822,Z 708.112,A -85,B 0,C 180,E1 -23443.951,E2 -23443.951} C_VEL
LIN {X 0,Y 209.475,Z 723.415,A -85,B 0,C 180,E1 -23443.276,E2 -23443.276} C_VEL
LIN {X 0,Y 208.117,Z 729.239,A -85,B 0,C 180,E1 -23443.379,E2 -23443.379} C_VEL
LIN {X 0,Y 205.202,Z 742.383,A -85,B 0,C 180,E1 -23444.187,E2 -23444.187} C_VEL
LIN {X 0,Y 201.754,Z 753.907,A -85,B 0,C 180,E1 -23445.14,E2 -23445.14} C_VEL
LIN {X 0,Y 197.501,Z 765.416,A -85,B 0,C 180,E1 -23446.415,E2 -23446.415} C_VEL
LIN {X 0,Y 192.193,Z 777.18,A -85,B 0,C 180,E1 -23448.138,E2 -23448.138} C_VEL
LIN {X 0,Y 186.696,Z 787.776,A -85,B 0,C 180,E1 -23450.213,E2 -23450.213} C_VEL
LIN {X 0,Y 181.547,Z 796.51,A -85,B 0,C 180,E1 -23452.432,E2 -23452.432} C_VEL
LIN {X 0,Y 175.953,Z 805.128,A -85,B 0,C 180,E1 -23455.308,E2 -23455.308} C_VEL
LIN {X 0,Y 170.857,Z 812.171,A -85,B 0,C 180,E1 -23458.369,E2 -23458.369} C_VEL
LIN {X 0,Y 165.835,Z 818.811,A -85,B 0,C 180,E1 -23462.215,E2 -23462.215} C_VEL
LIN {X 0,Y 162.797,Z 822.734,A -85,B 0,C 180,E1 -23465.231,E2 -23465.231} C_VEL
LIN {X 0,Y 159.401,Z 826.76,A -85,B 0,C 180,E1 -23469.347,E2 -23469.347} C_VEL
LIN {X 0,Y 156.692,Z 829.999,A -85,B 0,C 180,E1 -23474.389,E2 -23474.389} C_VEL
LIN {X 0,Y 155.437,Z 831.653,A -85,B 0,C 180,E1 -23479.581,E2 -23479.581} C_VEL
LIN {X 0,Y 155.464,Z 831.818,A -85,B 0,C 180,E1 -23484.813,E2 -23484.813} C_VEL
LIN {X 0,Y 155.669,Z 831.305,A -85,B 0,C 180,E1 -23487.412,E2 -23487.412} C_VEL
LIN {X 0,Y 156.076,Z 830.392,A -85,B 0,C 180,E1 -23490.322,E2 -23490.322} C_VEL
LIN {X 0,Y 155.431,Z 831.319,A -85,B 0,C 180,E1 -23495.188,E2 -23495.188} C_VEL
LIN {X 0,Y 155.439,Z 830.748,A -85,B 0,C 180,E1 -23500.419,E2 -23500.419} C_VEL
LIN {X 0,Y 155.915,Z 829.891,A -85,B 0,C 180,E1 -23503.025,E2 -23503.025} C_VEL
LIN {X 0,Y 157.917,Z 826.918,A -85,B 0,C 180,E1 -23508.151,E2 -23508.151} C_VEL
LIN {X 0,Y 160.283,Z 823.597,A -85,B 0,C 180,E1 -23511.882,E2 -23511.882} C_VEL
LIN {X 0,Y 163.248,Z 819.226,A -85,B 0,C 180,E1 -23515.499,E2 -23515.499} C_VEL
LIN {X 0,Y 166.959,Z 813.691,A -85,B 0,C 180,E1 -23518.952,E2 -23518.952} C_VEL
LIN {X 0,Y 171.426,Z 806.826,A -85,B 0,C 180,E1 -23522.205,E2 -23522.205} C_VEL
LIN {X 0,Y 176.526,Z 798.294,A -85,B 0,C 180,E1 -23525.259,E2 -23525.259} C_VEL
LIN {X 0,Y 181.127,Z 789.56,A -85,B 0,C 180,E1 -23527.67,E2 -23527.67} C_VEL
LIN {X 0,Y 186.19,Z 778.842,A -85,B 0,C 180,E1 -23529.917,E2 -23529.917} C_VEL
LIN {X 0,Y 190.547,Z 768.085,A -85,B 0,C 180,E1 -23531.597,E2 -23531.597} C_VEL
LIN {X 0,Y 194.518,Z 756.088,A -85,B 0,C 180,E1 -23532.996,E2 -23532.996} C_VEL
LIN {X 0,Y 197.653,Z 743.605,A -85,B 0,C 180,E1 -23534.073,E2 -23534.073} C_VEL
LIN {X 0,Y 199.882,Z 730.583,A -85,B 0,C 180,E1 -23534.836,E2 -23534.836} C_VEL
LIN {X 0,Y 201.245,Z 716.13,A -85,B 0,C 180,E1 -23535.369,E2 -23535.369} C_VEL
LIN {X 0,Y 202.621,Z 695.672,A -85,B 0,C 180,E1 -23536.028,E2 -23536.028} C_VEL
LIN {X 0,Y 201.942,Z 677.138,A -85,B 0,C 180,E1 -23537.315,E2 -23537.315} C_VEL
LIN {X 0,Y 198.565,Z 665.908,A -85,B 0,C 180,E1 -23539.264,E2 -23539.264} C_VEL
LIN {X 0,Y 193.649,Z 657.184,A -85,B 0,C 180,E1 -23541.905,E2 -23541.905} C_VEL
LIN {X 0,Y 188.681,Z 649.086,A -85,B 0,C 180,E1 -23544.889,E2 -23544.889} C_VEL
LIN {X 0,Y 184.425,Z 643.064,A -85,B 0,C 180,E1 -23547.757,E2 -23547.757} C_VEL
LIN {X 0,Y 181.009,Z 638.53,A -85,B 0,C 180,E1 -23550.376,E2 -23550.376} C_VEL
LIN {X 0,Y 178.281,Z 635.018,A -85,B 0,C 180,E1 -23552.744,E2 -23552.744} C_VEL
LIN {X 0,Y 177.452,Z 633.832,A -85,B 0,C 180,E1 -23553.541,E2 -23553.541} C_VEL
LIN {X 0,Y 174.757,Z 631.015,A -85,B 0,C 180,E1 -23556.287,E2 -23556.287} C_VEL
LIN {X 0,Y 173.649,Z 628.791,A -85,B 0,C 180,E1 -23557.71,E2 -23557.71} C_VEL
LIN {X 0,Y 170.988,Z 626.792,A -85,B 0,C 180,E1 -23561.27,E2 -23561.27} C_VEL
LIN {X 0,Y 169.277,Z 623.476,A -85,B 0,C 180,E1 -23564.768,E2 -23564.768} C_VEL
LIN {X 0,Y 168.953,Z 623.012,A -85,B 0,C 180,E1 -23565.547,E2 -23565.547} C_VEL
LIN {X 0,Y 167.058,Z 622.011,A -85,B 0,C 180,E1 -23572.749,E2 -23572.749} C_VEL
LIN {X 0,Y 167.761,Z 622.114,A -85,B 0,C 180,E1 -23580,E2 -23580} C_VEL
LIN {X 0,Y 169.475,Z 623.21,A -85,B 0,C 180,E1 -23584.512,E2 -23584.512} C_VEL
LIN {X 0,Y 170.768,Z 626.091,A -85,B 0,C 180,E1 -23587.241,E2 -23587.241} C_VEL
LIN {X 0,Y 173.373,Z 628.461,A -85,B 0,C 180,E1 -23590.904,E2 -23590.904} C_VEL
LIN {X 0,Y 173.9,Z 629.136,A -85,B 0,C 180,E1 -23591.56,E2 -23591.56} C_VEL
LIN {X 0,Y 176.036,Z 632.492,A -85,B 0,C 180,E1 -23594.044,E2 -23594.044} C_VEL
LIN {X 0,Y 178.022,Z 634.431,A -85,B 0,C 180,E1 -23595.941,E2 -23595.941} C_VEL
LIN {X 0,Y 180.484,Z 637.938,A -85,B 0,C 180,E1 -23598.151,E2 -23598.151} C_VEL
LIN {X 0,Y 182.031,Z 639.704,A -85,B 0,C 180,E1 -23599.379,E2 -23599.379} C_VEL
LIN {X 0,Y 185.75,Z 644.901,A -85,B 0,C 180,E1 -23602.129,E2 -23602.129} C_VEL
LIN {X 0,Y 188.58,Z 648.926,A -85,B 0,C 180,E1 -23604.001,E2 -23604.001} C_VEL
LIN {X 0,Y 193.423,Z 656.175,A -85,B 0,C 180,E1 -23606.876,E2 -23606.876} C_VEL
LIN {X 0,Y 198.712,Z 664.802,A -85,B 0,C 180,E1 -23609.68,E2 -23609.68} C_VEL
LIN {X 0,Y 204.126,Z 674.914,A -85,B 0,C 180,E1 -23612.29,E2 -23612.29} C_VEL
LIN {X 0,Y 204.317,Z 675.325,A -85,B 0,C 180,E1 -23612.379,E2 -23612.379} C_VEL
LIN {X 0,Y 202.352,Z 704.75,A -85,B 0,C 180,E1 -23613.424,E2 -23613.424} C_VEL
LIN {X 0,Y 200.704,Z 717.036,A -85,B 0,C 180,E1 -23614.15,E2 -23614.15} C_VEL
LIN {X 0,Y 198.094,Z 730.128,A -85,B 0,C 180,E1 -23615.316,E2 -23615.316} C_VEL
LIN {X 0,Y 195.055,Z 741.564,A -85,B 0,C 180,E1 -23616.71,E2 -23616.71} C_VEL
LIN {X 0,Y 191.457,Z 752.056,A -85,B 0,C 180,E1 -23618.359,E2 -23618.359} C_VEL
LIN {X 0,Y 187.113,Z 762.55,A -85,B 0,C 180,E1 -23620.485,E2 -23620.485} C_VEL
LIN {X 0,Y 182.463,Z 772.058,A -85,B 0,C 180,E1 -23622.961,E2 -23622.961} C_VEL
LIN {X 0,Y 177.36,Z 781.095,A -85,B 0,C 180,E1 -23626.098,E2 -23626.098} C_VEL
LIN {X 0,Y 172.716,Z 788.302,A -85,B 0,C 180,E1 -23629.38,E2 -23629.38} C_VEL
LIN {X 0,Y 168.371,Z 794.219,A -85,B 0,C 180,E1 -23632.993,E2 -23632.993} C_VEL
LIN {X 0,Y 164.994,Z 798.331,A -85,B 0,C 180,E1 -23636.377,E2 -23636.377} C_VEL
LIN {X 0,Y 161.82,Z 801.718,A -85,B 0,C 180,E1 -23640.299,E2 -23640.299} C_VEL
LIN {X 0,Y 159.572,Z 803.755,A -85,B 0,C 180,E1 -23643.87,E2 -23643.87} C_VEL
LIN {X 0,Y 157.314,Z 805.185,A -85,B 0,C 180,E1 -23649.06,E2 -23649.06} C_VEL
LIN {X 0,Y 156.531,Z 805.265,A -85,B 0,C 180,E1 -23651.683,E2 -23651.683} C_VEL
LIN {X 0,Y 155.673,Z 804.207,A -85,B 0,C 180,E1 -23656.955,E2 -23656.955} C_VEL
LIN {X 0,Y 155.625,Z 803.074,A -85,B 0,C 180,E1 -23659.593,E2 -23659.593} C_VEL
LIN {X 0,Y 155.844,Z 801.085,A -85,B 0,C 180,E1 -23662.805,E2 -23662.805} C_VEL
LIN {X 0,Y 156.741,Z 797.061,A -85,B 0,C 180,E1 -23667.43,E2 -23667.43} C_VEL
LIN {X 0,Y 157.892,Z 792.471,A -85,B 0,C 180,E1 -23671.275,E2 -23671.275} C_VEL
LIN {X 0,Y 159.889,Z 785.547,A -85,B 0,C 180,E1 -23675.676,E2 -23675.676} C_VEL
LIN {X 0,Y 162.197,Z 778.038,A -85,B 0,C 180,E1 -23679.351,E2 -23679.351} C_VEL
LIN {X 0,Y 165.089,Z 768.575,A -85,B 0,C 180,E1 -23682.914,E2 -23682.914} C_VEL
LIN {X 0,Y 167.706,Z 758.873,A -85,B 0,C 180,E1 -23685.806,E2 -23685.806} C_VEL
LIN {X 0,Y 169.34,Z 752.428,A -85,B 0,C 180,E1 -23687.364,E2 -23687.364} C_VEL
LIN {X 0,Y 167.606,Z 750.822,A -85,B 0,C 180,E1 -23688.108,E2 -23688.108} C_VEL
LIN {X 0,Y 167.427,Z 750.454,A -85,B 0,C 180,E1 -23688.242,E2 -23688.242} C_VEL
LIN {X 0,Y 164.908,Z 761.468,A -85,B 0,C 180,E1 -23690.986,E2 -23690.986} C_VEL
LIN {X 0,Y 162.519,Z 771.232,A -85,B 0,C 180,E1 -23694.1,E2 -23694.1} C_VEL
LIN {X 0,Y 160.056,Z 780.654,A -85,B 0,C 180,E1 -23697.896,E2 -23697.896} C_VEL
LIN {X 0,Y 158.384,Z 787.517,A -85,B 0,C 180,E1 -23701.424,E2 -23701.424} C_VEL
LIN {X 0,Y 156.92,Z 793.912,A -85,B 0,C 180,E1 -23705.607,E2 -23705.607} C_VEL
LIN {X 0,Y 155.886,Z 799.005,A -85,B 0,C 180,E1 -23709.965,E2 -23709.965} C_VEL
LIN {X 0,Y 155.523,Z 802.243,A -85,B 0,C 180,E1 -23713.695,E2 -23713.695} C_VEL
LIN {X 0,Y 155.605,Z 804.547,A -85,B 0,C 180,E1 -23717.353,E2 -23717.353} C_VEL
LIN {X 0,Y 156.176,Z 806.034,A -85,B 0,C 180,E1 -23720.949,E2 -23720.949} C_VEL
LIN {X 0,Y 157.168,Z 806.734,A -85,B 0,C 180,E1 -23724.457,E2 -23724.457} C_VEL
LIN {X 0,Y 158.607,Z 806.681,A -85,B 0,C 180,E1 -23727.878,E2 -23727.878} C_VEL
LIN {X 0,Y 160.451,Z 805.963,A -85,B 0,C 180,E1 -23731.196,E2 -23731.196} C_VEL
LIN {X 0,Y 163.07,Z 804.308,A -85,B 0,C 180,E1 -23734.828,E2 -23734.828} C_VEL
LIN {X 0,Y 167.33,Z 800.642,A -85,B 0,C 180,E1 -23739.462,E2 -23739.462} C_VEL
LIN {X 0,Y 171.962,Z 795.911,A -85,B 0,C 180,E1 -23743.376,E2 -23743.376} C_VEL
LIN {X 0,Y 176.795,Z 790.211,A -85,B 0,C 180,E1 -23746.764,E2 -23746.764} C_VEL
LIN {X 0,Y 182.164,Z 782.9,A -85,B 0,C 180,E1 -23750.002,E2 -23750.002} C_VEL
LIN {X 0,Y 187.064,Z 775.398,A -85,B 0,C 180,E1 -23752.519,E2 -23752.519} C_VEL
LIN {X 0,Y 192.479,Z 765.682,A -85,B 0,C 180,E1 -23755.067,E2 -23755.067} C_VEL
LIN {X 0,Y 197.049,Z 756.129,A -85,B 0,C 180,E1 -23757.003,E2 -23757.003} C_VEL
LIN {X 0,Y 201.475,Z 745.087,A -85,B 0,C 180,E1 -23758.752,E2 -23758.752} C_VEL
LIN {X 0,Y 205.323,Z 733.053,A -85,B 0,C 180,E1 -23760.212,E2 -23760.212} C_VEL
LIN {X 0,Y 208.439,Z 719.856,A -85,B 0,C 180,E1 -23761.408,E2 -23761.408} C_VEL
LIN {X 0,Y 210.503,Z 707.194,A -85,B 0,C 180,E1 -23762.216,E2 -23762.216} C_VEL
LIN {X 0,Y 213.431,Z 679.405,A -85,B 0,C 180,E1 -23763.347,E2 -23763.347} C_VEL
LIN {X 0,Y 209.084,Z 670.195,A -85,B 0,C 180,E1 -23767.032,E2 -23767.032} C_VEL
LIN {X 0,Y 207.062,Z 666.963,A -85,B 0,C 180,E1 -23769.039,E2 -23769.039} C_VEL
LIN {X 0,Y 204.731,Z 662.948,A -85,B 0,C 180,E1 -23771.886,E2 -23771.886} C_VEL
LIN {X 0,Y 202.739,Z 659.711,A -85,B 0,C 180,E1 -23775.191,E2 -23775.191} C_VEL
LIN {X 0,Y 202.339,Z 658.952,A -85,B 0,C 180,E1 -23776.133,E2 -23776.133} C_VEL
LIN {X 0,Y 201.018,Z 658.036,A -85,B 0,C 180,E1 -23780.464,E2 -23780.464} C_VEL
LIN {X 0,Y 200.845,Z 658.585,A -85,B 0,C 180,E1 -23783.451,E2 -23783.451} C_VEL
LIN {X 0,Y 201.316,Z 660.639,A -85,B 0,C 180,E1 -23786.823,E2 -23786.823} C_VEL
LIN {X 0,Y 203.231,Z 665.341,A -85,B 0,C 180,E1 -23791.39,E2 -23791.39} C_VEL
LIN {X 0,Y 205.583,Z 671.433,A -85,B 0,C 180,E1 -23794.917,E2 -23794.917} C_VEL
LIN {X 0,Y 207.593,Z 676.887,A -85,B 0,C 180,E1 -23797.298,E2 -23797.298} C_VEL
LIN {X 0,Y 209.342,Z 681.734,A -85,B 0,C 180,E1 -23799.035,E2 -23799.035} C_VEL
LIN {X 0,Y 211.642,Z 689.322,A -85,B 0,C 180,E1 -23801.213,E2 -23801.213} C_VEL
LIN {X 0,Y 211.752,Z 694.278,A -85,B 0,C 180,E1 -23801.737,E2 -23801.737} C_VEL
LIN {X 0,Y 211.485,Z 702.098,A -85,B 0,C 180,E1 -23802.323,E2 -23802.323} C_VEL
LIN {X 0,Y 208.61,Z 726.273,A -85,B 0,C 180,E1 -23803.24,E2 -23803.24} C_VEL
LIN {X 0,Y 208.117,Z 729.239,A -85,B 0,C 180,E1 -23803.379,E2 -23803.379} C_VEL
LIN {X 0,Y 207.19,Z 733.038,A -85,B 0,C 180,E1 -23803.495,E2 -23803.495} C_VEL
LIN {X 0,Y 204.46,Z 740.474,A -85,B 0,C 180,E1 -23803.461,E2 -23803.461} C_VEL
LIN {X 0,Y 199.431,Z 751.303,A -85,B 0,C 180,E1 -23803.42,E2 -23803.42} C_VEL
LIN {X 0,Y 197.078,Z 756.654,A -85,B 0,C 180,E1 -23803.701,E2 -23803.701} C_VEL
LIN {X 0,Y 196.39,Z 758.373,A -85,B 0,C 180,E1 -23803.864,E2 -23803.864} C_VEL
LIN {X 0,Y 191.891,Z 769.114,A -85,B 0,C 180,E1 -23805.169,E2 -23805.169} C_VEL
LIN {X 0,Y 186.457,Z 780.02,A -85,B 0,C 180,E1 -23806.909,E2 -23806.909} C_VEL
LIN {X 0,Y 180.248,Z 790.768,A -85,B 0,C 180,E1 -23809.226,E2 -23809.226} C_VEL
LIN {X 0,Y 174.015,Z 800.34,A -85,B 0,C 180,E1 -23811.983,E2 -23811.983} C_VEL
LIN {X 0,Y 168.316,Z 808.122,A -85,B 0,C 180,E1 -23814.962,E2 -23814.962} C_VEL
LIN {X 0,Y 162.49,Z 815.436,A -85,B 0,C 180,E1 -23818.734,E2 -23818.734} C_VEL
LIN {X 0,Y 158.262,Z 820.424,A -85,B 0,C 180,E1 -23822.208,E2 -23822.208} C_VEL
LIN {X 0,Y 154.785,Z 824.398,A -85,B 0,C 180,E1 -23825.881,E2 -23825.881} C_VEL
LIN {X 0,Y 152.751,Z 826.525,A -85,B 0,C 180,E1 -23828.404,E2 -23828.404} C_VEL
LIN {X 0,Y 151.144,Z 828.247,A -85,B 0,C 180,E1 -23831.005,E2 -23831.005} C_VEL
LIN {X 0,Y 148.951,Z 830.479,A -85,B 0,C 180,E1 -23836.355,E2 -23836.355} C_VEL
LIN {X 0,Y 148.239,Z 831.253,A -85,B 0,C 180,E1 -23841.823,E2 -23841.823} C_VEL
LIN {X 0,Y 148.384,Z 831.069,A -85,B 0,C 180,E1 -23844.565,E2 -23844.565} C_VEL
LIN {X 0,Y 149.036,Z 829.558,A -85,B 0,C 180,E1 -23850,E2 -23850} C_VEL
LIN {X 0,Y 148.556,Z 830.339,A -85,B 0,C 180,E1 -23852.712,E2 -23852.712} C_VEL
LIN {X 0,Y 148.325,Z 830.701,A -85,B 0,C 180,E1 -23855.714,E2 -23855.714} C_VEL
LIN {X 0,Y 148.43,Z 830.183,A -85,B 0,C 180,E1 -23860.917,E2 -23860.917} C_VEL
LIN {X 0,Y 148.963,Z 829.359,A -85,B 0,C 180,E1 -23863.644,E2 -23863.644} C_VEL
LIN {X 0,Y 149.841,Z 828.12,A -85,B 0,C 180,E1 -23866.344,E2 -23866.344} C_VEL
LIN {X 0,Y 152.722,Z 824.407,A -85,B 0,C 180,E1 -23871.601,E2 -23871.601} C_VEL
LIN {X 0,Y 155.925,Z 820.162,A -85,B 0,C 180,E1 -23875.649,E2 -23875.649} C_VEL
LIN {X 0,Y 159.34,Z 815.409,A -85,B 0,C 180,E1 -23879.023,E2 -23879.023} C_VEL
LIN {X 0,Y 163.823,Z 809.107,A -85,B 0,C 180,E1 -23882.428,E2 -23882.428} C_VEL
LIN {X 0,Y 168.92,Z 801.263,A -85,B 0,C 180,E1 -23885.624,E2 -23885.624} C_VEL
LIN {X 0,Y 173.647,Z 793.296,A -85,B 0,C 180,E1 -23888.112,E2 -23888.112} C_VEL
LIN {X 0,Y 178.738,Z 783.602,A -85,B 0,C 180,E1 -23890.449,E2 -23890.449} C_VEL
LIN {X 0,Y 183.056,Z 774.131,A -85,B 0,C 180,E1 -23892.21,E2 -23892.21} C_VEL
LIN {X 0,Y 187.045,Z 763.981,A -85,B 0,C 180,E1 -23893.662,E2 -23893.662} C_VEL
LIN {X 0,Y 190.899,Z 751.905,A -85,B 0,C 180,E1 -23894.941,E2 -23894.941} C_VEL
LIN {X 0,Y 194.01,Z 738.64,A -85,B 0,C 180,E1 -23895.957,E2 -23895.957} C_VEL
LIN {X 0,Y 195.979,Z 725.918,A -85,B 0,C 180,E1 -23896.598,E2 -23896.598} C_VEL
LIN {X 0,Y 198.147,Z 696.573,A -85,B 0,C 180,E1 -23897.589,E2 -23897.589} C_VEL
LIN {X 0,Y 197.668,Z 679.823,A -85,B 0,C 180,E1 -23898.772,E2 -23898.772} C_VEL
LIN {X 0,Y 194.844,Z 670.283,A -85,B 0,C 180,E1 -23900.519,E2 -23900.519} C_VEL
LIN {X 0,Y 190.414,Z 662.277,A -85,B 0,C 180,E1 -23903.064,E2 -23903.064} C_VEL
LIN {X 0,Y 185.906,Z 654.65,A -85,B 0,C 180,E1 -23905.953,E2 -23905.953} C_VEL
LIN {X 0,Y 182.099,Z 649.143,A -85,B 0,C 180,E1 -23908.68,E2 -23908.68} C_VEL
LIN {X 0,Y 178.943,Z 644.81,A -85,B 0,C 180,E1 -23911.241,E2 -23911.241} C_VEL
LIN {X 0,Y 176.248,Z 641.077,A -85,B 0,C 180,E1 -23913.745,E2 -23913.745} C_VEL
LIN {X 0,Y 172.959,Z 637.19,A -85,B 0,C 180,E1 -23917.293,E2 -23917.293} C_VEL
LIN {X 0,Y 172.115,Z 635.55,A -85,B 0,C 180,E1 -23918.439,E2 -23918.439} C_VEL
LIN {X 0,Y 169.545,Z 633.313,A -85,B 0,C 180,E1 -23922.166,E2 -23922.166} C_VEL
LIN {X 0,Y 167.967,Z 630.026,A -85,B 0,C 180,E1 -23925.77,E2 -23925.77} C_VEL
LIN {X 0,Y 166.185,Z 629.063,A -85,B 0,C 180,E1 -23932.711,E2 -23932.711} C_VEL
LIN {X 0,Y 166.884,Z 629.183,A -85,B 0,C 180,E1 -23940,E2 -23940} C_VEL
LIN {X 0,Y 168.344,Z 630.203,A -85,B 0,C 180,E1 -23944.02,E2 -23944.02} C_VEL
LIN {X 0,Y 169.662,Z 633.078,A -85,B 0,C 180,E1 -23946.914,E2 -23946.914} C_VEL
LIN {X 0,Y 172.321,Z 635.676,A -85,B 0,C 180,E1 -23950.773,E2 -23950.773} C_VEL
LIN {X 0,Y 174.603,Z 639.261,A -85,B 0,C 180,E1 -23953.549,E2 -23953.549} C_VEL
LIN {X 0,Y 176.239,Z 640.951,A -85,B 0,C 180,E1 -23955.189,E2 -23955.189} C_VEL
LIN {X 0,Y 178.908,Z 644.741,A -85,B 0,C 180,E1 -23957.678,E2 -23957.678} C_VEL
LIN {X 0,Y 180.112,Z 646.249,A -85,B 0,C 180,E1 -23958.683,E2 -23958.683} C_VEL
LIN {X 0,Y 183.51,Z 651.149,A -85,B 0,C 180,E1 -23961.32,E2 -23961.32} C_VEL
LIN {X 0,Y 186.468,Z 655.533,A -85,B 0,C 180,E1 -23963.377,E2 -23963.377} C_VEL
LIN {X 0,Y 191.02,Z 662.622,A -85,B 0,C 180,E1 -23966.2,E2 -23966.2} C_VEL
LIN {X 0,Y 195.791,Z 670.75,A -85,B 0,C 180,E1 -23968.858,E2 -23968.858} C_VEL
LIN {X 0,Y 199.76,Z 678.31,A -85,B 0,C 180,E1 -23970.892,E2 -23970.892} C_VEL
LIN {X 0,Y 197.805,Z 705.83,A -85,B 0,C 180,E1 -23971.884,E2 -23971.884} C_VEL
LIN {X 0,Y 196.023,Z 718.317,A -85,B 0,C 180,E1 -23972.648,E2 -23972.648} C_VEL
LIN {X 0,Y 193.395,Z 730.82,A -85,B 0,C 180,E1 -23973.772,E2 -23973.772} C_VEL
LIN {X 0,Y 190.226,Z 742.238,A -85,B 0,C 180,E1 -23975.175,E2 -23975.175} C_VEL
LIN {X 0,Y 186.54,Z 752.586,A -85,B 0,C 180,E1 -23976.814,E2 -23976.814} C_VEL
LIN {X 0,Y 182.371,Z 762.283,A -85,B 0,C 180,E1 -23978.768,E2 -23978.768} C_VEL
LIN {X 0,Y 177.561,Z 771.824,A -85,B 0,C 180,E1 -23981.235,E2 -23981.235} C_VEL
LIN {X 0,Y 173.116,Z 779.535,A -85,B 0,C 180,E1 -23983.808,E2 -23983.808} C_VEL
LIN {X 0,Y 168.001,Z 787.27,A -85,B 0,C 180,E1 -23987.174,E2 -23987.174} C_VEL
LIN {X 0,Y 163.349,Z 793.447,A -85,B 0,C 180,E1 -23990.754,E2 -23990.754} C_VEL
LIN {X 0,Y 158.939,Z 798.647,A -85,B 0,C 180,E1 -23994.913,E2 -23994.913} C_VEL
LIN {X 0,Y 155.233,Z 802.369,A -85,B 0,C 180,E1 -23999.34,E2 -23999.34} C_VEL
LIN {X 0,Y 153.052,Z 804.237,A -85,B 0,C 180,E1 -24002.666,E2 -24002.666} C_VEL
LIN {X 0,Y 150.533,Z 805.744,A -85,B 0,C 180,E1 -24008.069,E2 -24008.069} C_VEL
LIN {X 0,Y 149.66,Z 805.897,A -85,B 0,C 180,E1 -24010.81,E2 -24010.81} C_VEL
LIN {X 0,Y 149.028,Z 805.602,A -85,B 0,C 180,E1 -24013.564,E2 -24013.564} C_VEL
LIN {X 0,Y 148.552,Z 803.838,A -85,B 0,C 180,E1 -24019.092,E2 -24019.092} C_VEL
LIN {X 0,Y 148.762,Z 801.684,A -85,B 0,C 180,E1 -24022.798,E2 -24022.798} C_VEL
LIN {X 0,Y 149.616,Z 797.98,A -85,B 0,C 180,E1 -24027.308,E2 -24027.308} C_VEL
LIN {X 0,Y 150.777,Z 793.494,A -85,B 0,C 180,E1 -24031.335,E2 -24031.335} C_VEL
LIN {X 0,Y 152.841,Z 786.674,A -85,B 0,C 180,E1 -24035.938,E2 -24035.938} C_VEL
LIN {X 0,Y 155.206,Z 779.293,A -85,B 0,C 180,E1 -24039.776,E2 -24039.776} C_VEL
LIN {X 0,Y 157.636,Z 771.741,A -85,B 0,C 180,E1 -24042.88,E2 -24042.88} C_VEL
LIN {X 0,Y 160.395,Z 762.538,A -85,B 0,C 180,E1 -24045.893,E2 -24045.893} C_VEL
LIN {X 0,Y 161.522,Z 758.305,A -85,B 0,C 180,E1 -24047.079,E2 -24047.079} C_VEL
LIN {X 0,Y 160.932,Z 756.329,A -85,B 0,C 180,E1 -24047.8,E2 -24047.8} C_VEL
LIN {X 0,Y 159.735,Z 755.03,A -85,B 0,C 180,E1 -24048.476,E2 -24048.476} C_VEL
LIN {X 0,Y 156.982,Z 766.266,A -85,B 0,C 180,E1 -24051.675,E2 -24051.675} C_VEL
LIN {X 0,Y 154.407,Z 775.944,A -85,B 0,C 180,E1 -24055.232,E2 -24055.232} C_VEL
LIN {X 0,Y 152.362,Z 783.646,A -85,B 0,C 180,E1 -24058.787,E2 -24058.787} C_VEL
LIN {X 0,Y 150.634,Z 790.694,A -85,B 0,C 180,E1 -24062.88,E2 -24062.88} C_VEL
LIN {X 0,Y 149.424,Z 796.119,A -85,B 0,C 180,E1 -24066.91,E2 -24066.91} C_VEL
LIN {X 0,Y 148.615,Z 800.772,A -85,B 0,C 180,E1 -24071.456,E2 -24071.456} C_VEL
LIN {X 0,Y 148.42,Z 803.675,A -85,B 0,C 180,E1 -24075.257,E2 -24075.257} C_VEL
LIN {X 0,Y 148.719,Z 805.762,A -85,B 0,C 180,E1 -24079.121,E2 -24079.121} C_VEL
LIN {X 0,Y 149.584,Z 807.015,A -85,B 0,C 180,E1 -24083.006,E2 -24083.006} C_VEL
LIN {X 0,Y 150.999,Z 807.465,A -85,B 0,C 180,E1 -24086.904,E2 -24086.904} C_VEL
LIN {X 0,Y 153.011,Z 807.076,A -85,B 0,C 180,E1 -24090.771,E2 -24090.771} C_VEL
LIN {X 0,Y 155.594,Z 805.808,A -85,B 0,C 180,E1 -24094.603,E2 -24094.603} C_VEL
LIN {X 0,Y 159.865,Z 802.758,A -85,B 0,C 180,E1 -24099.409,E2 -24099.409} C_VEL
LIN {X 0,Y 163.25,Z 799.806,A -85,B 0,C 180,E1 -24102.461,E2 -24102.461} C_VEL
LIN {X 0,Y 169.088,Z 793.9,A -85,B 0,C 180,E1 -24106.785,E2 -24106.785} C_VEL
LIN {X 0,Y 174.786,Z 787.088,A -85,B 0,C 180,E1 -24110.266,E2 -24110.266} C_VEL
LIN {X 0,Y 180.56,Z 779.176,A -85,B 0,C 180,E1 -24113.294,E2 -24113.294} C_VEL
LIN {X 0,Y 186.26,Z 770.082,A -85,B 0,C 180,E1 -24115.931,E2 -24115.931} C_VEL
LIN {X 0,Y 191.617,Z 760.009,A -85,B 0,C 180,E1 -24118.161,E2 -24118.161} C_VEL
LIN {X 0,Y 196.471,Z 749.159,A -85,B 0,C 180,E1 -24120,E2 -24120} C_VEL
LIN {X 0,Y 200.271,Z 738.65,A -85,B 0,C 180,E1 -24121.383,E2 -24121.383} C_VEL
LIN {X 0,Y 204.041,Z 725.247,A -85,B 0,C 180,E1 -24122.744,E2 -24122.744} C_VEL
LIN {X 0,Y 206.561,Z 712.64,A -85,B 0,C 180,E1 -24123.662,E2 -24123.662} C_VEL
LIN {X 0,Y 208.225,Z 699.697,A -85,B 0,C 180,E1 -24124.292,E2 -24124.292} C_VEL
LIN {X 0,Y 210.017,Z 683.355,A -85,B 0,C 180,E1 -24124.937,E2 -24124.937} C_VEL
LIN {X 0,Y 206.902,Z 676.18,A -85,B 0,C 180,E1 -24127.907,E2 -24127.907} C_VEL
LIN {X 0,Y 205.132,Z 673.335,A -85,B 0,C 180,E1 -24129.763,E2 -24129.763} C_VEL
LIN {X 0,Y 203.001,Z 669.448,A -85,B 0,C 180,E1 -24132.638,E2 -24132.638} C_VEL
LIN {X 0,Y 201.151,Z 665.955,A -85,B 0,C 180,E1 -24136.231,E2 -24136.231} C_VEL
LIN {X 0,Y 199.868,Z 665.058,A -85,B 0,C 180,E1 -24140.587,E2 -24140.587} C_VEL
LIN {X 0,Y 199.712,Z 665.714,A -85,B 0,C 180,E1 -24143.575,E2 -24143.575} C_VEL
LIN {X 0,Y 200.089,Z 667.654,A -85,B 0,C 180,E1 -24146.593,E2 -24146.593} C_VEL
LIN {X 0,Y 201.683,Z 671.953,A -85,B 0,C 180,E1 -24150.793,E2 -24150.793} C_VEL
LIN {X 0,Y 203.693,Z 677.772,A -85,B 0,C 180,E1 -24154.17,E2 -24154.17} C_VEL
LIN {X 0,Y 205.545,Z 683.209,A -85,B 0,C 180,E1 -24156.543,E2 -24156.543} C_VEL
LIN {X 0,Y 207.078,Z 687.959,A -85,B 0,C 180,E1 -24158.256,E2 -24158.256} C_VEL
LIN {X 0,Y 208.577,Z 693.664,A -85,B 0,C 180,E1 -24159.855,E2 -24159.855} C_VEL
LIN {X 0,Y 208.115,Z 703.757,A -85,B 0,C 180,E1 -24160.644,E2 -24160.644} C_VEL
LIN {X 0,Y 205.362,Z 725.471,A -85,B 0,C 180,E1 -24161.468,E2 -24161.468} C_VEL
LIN {X 0,Y 202.537,Z 738.965,A -85,B 0,C 180,E1 -24162.209,E2 -24162.209} C_VEL
LIN {X 0,Y 198.81,Z 751.58,A -85,B 0,C 180,E1 -24163.19,E2 -24163.19} C_VEL
LIN {X 0,Y 196.39,Z 758.373,A -85,B 0,C 180,E1 -24163.864,E2 -24163.864} C_VEL
LIN {X 0,Y 193.961,Z 763.585,A -85,B 0,C 180,E1 -24164.283,E2 -24164.283} C_VEL
LIN {X 0,Y 188.599,Z 771.844,A -85,B 0,C 180,E1 -24164.656,E2 -24164.656} C_VEL
LIN {X 0,Y 182.873,Z 779.71,A -85,B 0,C 180,E1 -24165.211,E2 -24165.211} C_VEL
LIN {X 0,Y 179.898,Z 784.207,A -85,B 0,C 180,E1 -24165.932,E2 -24165.932} C_VEL
LIN {X 0,Y 173.844,Z 793.603,A -85,B 0,C 180,E1 -24168.162,E2 -24168.162} C_VEL
LIN {X 0,Y 167.502,Z 802.467,A -85,B 0,C 180,E1 -24170.998,E2 -24170.998} C_VEL
LIN {X 0,Y 161.623,Z 809.719,A -85,B 0,C 180,E1 -24174.054,E2 -24174.054} C_VEL
LIN {X 0,Y 156.459,Z 815.669,A -85,B 0,C 180,E1 -24177.383,E2 -24177.383} C_VEL
LIN {X 0,Y 151.996,Z 820.48,A -85,B 0,C 180,E1 -24180.956,E2 -24180.956} C_VEL
LIN {X 0,Y 148.289,Z 824.264,A -85,B 0,C 180,E1 -24184.752,E2 -24184.752} C_VEL
LIN {X 0,Y 146.152,Z 826.264,A -85,B 0,C 180,E1 -24187.376,E2 -24187.376} C_VEL
LIN {X 0,Y 142.98,Z 829.087,A -85,B 0,C 180,E1 -24192.848,E2 -24192.848} C_VEL
LIN {X 0,Y 141.413,Z 830.446,A -85,B 0,C 180,E1 -24198.534,E2 -24198.534} C_VEL
LIN {X 0,Y 141.307,Z 830.268,A -85,B 0,C 180,E1 -24204.291,E2 -24204.291} C_VEL
LIN {X 0,Y 141.924,Z 828.718,A -85,B 0,C 180,E1 -24209.645,E2 -24209.645} C_VEL
LIN {X 0,Y 141.469,Z 829.663,A -85,B 0,C 180,E1 -24212.847,E2 -24212.847} C_VEL
LIN {X 0,Y 141.261,Z 830.073,A -85,B 0,C 180,E1 -24215.71,E2 -24215.71} C_VEL
LIN {X 0,Y 141.412,Z 829.615,A -85,B 0,C 180,E1 -24221.466,E2 -24221.466} C_VEL
LIN {X 0,Y 142.997,Z 827.636,A -85,B 0,C 180,E1 -24227.15,E2 -24227.15} C_VEL
LIN {X 0,Y 146.117,Z 823.989,A -85,B 0,C 180,E1 -24232.63,E2 -24232.63} C_VEL
LIN {X 0,Y 149.181,Z 820.216,A -85,B 0,C 180,E1 -24236.478,E2 -24236.478} C_VEL
LIN {X 0,Y 153.148,Z 815.132,A -85,B 0,C 180,E1 -24240.317,E2 -24240.317} C_VEL
LIN {X 0,Y 157.856,Z 808.911,A -85,B 0,C 180,E1 -24243.815,E2 -24243.815} C_VEL
LIN {X 0,Y 163.193,Z 801.201,A -85,B 0,C 180,E1 -24247.078,E2 -24247.078} C_VEL
LIN {X 0,Y 169.128,Z 791.575,A -85,B 0,C 180,E1 -24250.096,E2 -24250.096} C_VEL
LIN {X 0,Y 174.487,Z 781.656,A -85,B 0,C 180,E1 -24252.426,E2 -24252.426} C_VEL
LIN {X 0,Y 179.669,Z 770.455,A -85,B 0,C 180,E1 -24254.362,E2 -24254.362} C_VEL
LIN {X 0,Y 183.838,Z 759.525,A -85,B 0,C 180,E1 -24255.789,E2 -24255.789} C_VEL
LIN {X 0,Y 187.488,Z 747.432,A -85,B 0,C 180,E1 -24256.965,E2 -24256.965} C_VEL
LIN {X 0,Y 190.35,Z 734.178,A -85,B 0,C 180,E1 -24257.859,E2 -24257.859} C_VEL
LIN {X 0,Y 192.102,Z 721.23,A -85,B 0,C 180,E1 -24258.424,E2 -24258.424} C_VEL
LIN {X 0,Y 193.847,Z 697.582,A -85,B 0,C 180,E1 -24259.206,E2 -24259.206} C_VEL
LIN {X 0,Y 193.482,Z 682.345,A -85,B 0,C 180,E1 -24260.323,E2 -24260.323} C_VEL
LIN {X 0,Y 191.393,Z 675.025,A -85,B 0,C 180,E1 -24261.726,E2 -24261.726} C_VEL
LIN {X 0,Y 187.321,Z 667.42,A -85,B 0,C 180,E1 -24264.227,E2 -24264.227} C_VEL
LIN {X 0,Y 183.366,Z 660.49,A -85,B 0,C 180,E1 -24266.932,E2 -24266.932} C_VEL
LIN {X 0,Y 179.863,Z 655.248,A -85,B 0,C 180,E1 -24269.596,E2 -24269.596} C_VEL
LIN {X 0,Y 177.022,Z 651.22,A -85,B 0,C 180,E1 -24272.032,E2 -24272.032} C_VEL
LIN {X 0,Y 174.102,Z 647.09,A -85,B 0,C 180,E1 -24274.922,E2 -24274.922} C_VEL
LIN {X 0,Y 171.417,Z 643.776,A -85,B 0,C 180,E1 -24278.03,E2 -24278.03} C_VEL
LIN {X 0,Y 170.655,Z 642.337,A -85,B 0,C 180,E1 -24279.116,E2 -24279.116} C_VEL
LIN {X 0,Y 168.112,Z 639.761,A -85,B 0,C 180,E1 -24283.153,E2 -24283.153} C_VEL
LIN {X 0,Y 166.975,Z 637.118,A -85,B 0,C 180,E1 -24285.994,E2 -24285.994} C_VEL
LIN {X 0,Y 165.316,Z 636.094,A -85,B 0,C 180,E1 -24292.673,E2 -24292.673} C_VEL
LIN {X 0,Y 166.006,Z 636.248,A -85,B 0,C 180,E1 -24300,E2 -24300} C_VEL
LIN {X 0,Y 167.208,Z 637.086,A -85,B 0,C 180,E1 -24303.46,E2 -24303.46} C_VEL
LIN {X 0,Y 168.647,Z 640.132,A -85,B 0,C 180,E1 -24306.731,E2 -24306.731} C_VEL
LIN {X 0,Y 170.909,Z 642.463,A -85,B 0,C 180,E1 -24310.164,E2 -24310.164} C_VEL
LIN {X 0,Y 173.249,Z 646.152,A -85,B 0,C 180,E1 -24313.126,E2 -24313.126} C_VEL
LIN {X 0,Y 174.59,Z 647.644,A -85,B 0,C 180,E1 -24314.534,E2 -24314.534} C_VEL
LIN {X 0,Y 177.346,Z 651.529,A -85,B 0,C 180,E1 -24317.198,E2 -24317.198} C_VEL
LIN {X 0,Y 181.231,Z 657.218,A -85,B 0,C 180,E1 -24320.427,E2 -24320.427} C_VEL
LIN {X 0,Y 185.586,Z 663.919,A -85,B 0,C 180,E1 -24323.546,E2 -24323.546} C_VEL
LIN {X 0,Y 191.182,Z 673.378,A -85,B 0,C 180,E1 -24327.013,E2 -24327.013} C_VEL
LIN {X 0,Y 195.315,Z 681.273,A -85,B 0,C 180,E1 -24329.322,E2 -24329.322} C_VEL
LIN {X 0,Y 193.485,Z 706.203,A -85,B 0,C 180,E1 -24330.243,E2 -24330.243} C_VEL
LIN {X 0,Y 191.619,Z 718.831,A -85,B 0,C 180,E1 -24331.01,E2 -24331.01} C_VEL
LIN {X 0,Y 188.843,Z 731.51,A -85,B 0,C 180,E1 -24332.151,E2 -24332.151} C_VEL
LIN {X 0,Y 185.546,Z 742.913,A -85,B 0,C 180,E1 -24333.563,E2 -24333.563} C_VEL
LIN {X 0,Y 181.703,Z 753.247,A -85,B 0,C 180,E1 -24335.208,E2 -24335.208} C_VEL
LIN {X 0,Y 176.915,Z 763.858,A -85,B 0,C 180,E1 -24337.393,E2 -24337.393} C_VEL
LIN {X 0,Y 171.841,Z 773.351,A -85,B 0,C 180,E1 -24339.931,E2 -24339.931} C_VEL
LIN {X 0,Y 166.806,Z 781.495,A -85,B 0,C 180,E1 -24342.808,E2 -24342.808} C_VEL
LIN {X 0,Y 161.875,Z 788.459,A -85,B 0,C 180,E1 -24346.001,E2 -24346.001} C_VEL
LIN {X 0,Y 157.359,Z 794.106,A -85,B 0,C 180,E1 -24349.399,E2 -24349.399} C_VEL
LIN {X 0,Y 153.024,Z 798.944,A -85,B 0,C 180,E1 -24353.342,E2 -24353.342} C_VEL
LIN {X 0,Y 148.692,Z 803.024,A -85,B 0,C 180,E1 -24358.296,E2 -24358.296} C_VEL
LIN {X 0,Y 146.604,Z 804.708,A -85,B 0,C 180,E1 -24361.355,E2 -24361.355} C_VEL
LIN {X 0,Y 145.04,Z 805.713,A -85,B 0,C 180,E1 -24364.145,E2 -24364.145} C_VEL
LIN {X 0,Y 142.83,Z 806.503,A -85,B 0,C 180,E1 -24369.853,E2 -24369.853} C_VEL
LIN {X 0,Y 142.098,Z 806.275,A -85,B 0,C 180,E1 -24372.738,E2 -24372.738} C_VEL
LIN {X 0,Y 141.485,Z 804.585,A -85,B 0,C 180,E1 -24378.54,E2 -24378.54} C_VEL
LIN {X 0,Y 141.687,Z 802.296,A -85,B 0,C 180,E1 -24382.77,E2 -24382.77} C_VEL
LIN {X 0,Y 142.467,Z 798.884,A -85,B 0,C 180,E1 -24387.172,E2 -24387.172} C_VEL
LIN {X 0,Y 143.668,Z 794.485,A -85,B 0,C 180,E1 -24391.402,E2 -24391.402} C_VEL
LIN {X 0,Y 145.8,Z 787.802,A -85,B 0,C 180,E1 -24396.226,E2 -24396.226} C_VEL
LIN {X 0,Y 148.233,Z 780.531,A -85,B 0,C 180,E1 -24400.241,E2 -24400.241} C_VEL
LIN {X 0,Y 150.733,Z 773.108,A -85,B 0,C 180,E1 -24403.481,E2 -24403.481} C_VEL
LIN {X 0,Y 153.633,Z 764.118,A -85,B 0,C 180,E1 -24406.613,E2 -24406.613} C_VEL
LIN {X 0,Y 154.18,Z 762.06,A -85,B 0,C 180,E1 -24407.234,E2 -24407.234} C_VEL
LIN {X 0,Y 152.114,Z 759.164,A -85,B 0,C 180,E1 -24408.662,E2 -24408.662} C_VEL
LIN {X 0,Y 148.965,Z 770.982,A -85,B 0,C 180,E1 -24412.539,E2 -24412.539} C_VEL
LIN {X 0,Y 146.454,Z 780.003,A -85,B 0,C 180,E1 -24416.351,E2 -24416.351} C_VEL
LIN {X 0,Y 144.304,Z 788.241,A -85,B 0,C 180,E1 -24420.793,E2 -24420.793} C_VEL
LIN {X 0,Y 142.883,Z 794.039,A -85,B 0,C 180,E1 -24424.787,E2 -24424.787} C_VEL
LIN {X 0,Y 141.906,Z 798.662,A -85,B 0,C 180,E1 -24428.819,E2 -24428.819} C_VEL
LIN {X 0,Y 141.343,Z 803.171,A -85,B 0,C 180,E1 -24434.115,E2 -24434.115} C_VEL
LIN {X 0,Y 141.753,Z 806.41,A -85,B 0,C 180,E1 -24439.87,E2 -24439.87} C_VEL
LIN {X 0,Y 142.692,Z 807.637,A -85,B 0,C 180,E1 -24443.769,E2 -24443.769} C_VEL
LIN {X 0,Y 144.116,Z 808.137,A -85,B 0,C 180,E1 -24447.559,E2 -24447.559} C_VEL
LIN {X 0,Y 146.054,Z 807.939,A -85,B 0,C 180,E1 -24451.237,E2 -24451.237} C_VEL
LIN {X 0,Y 148.403,Z 807.017,A -85,B 0,C 180,E1 -24454.772,E2 -24454.772} C_VEL
LIN {X 0,Y 152.897,Z 804.355,A -85,B 0,C 180,E1 -24459.858,E2 -24459.858} C_VEL
LIN {X 0,Y 156.665,Z 801.448,A -85,B 0,C 180,E1 -24463.289,E2 -24463.289} C_VEL
LIN {X 0,Y 162.394,Z 796.208,A -85,B 0,C 180,E1 -24467.503,E2 -24467.503} C_VEL
LIN {X 0,Y 167.874,Z 790.417,A -85,B 0,C 180,E1 -24470.854,E2 -24470.854} C_VEL
LIN {X 0,Y 172.957,Z 784.234,A -85,B 0,C 180,E1 -24473.585,E2 -24473.585} C_VEL
LIN {X 0,Y 178.879,Z 776.054,A -85,B 0,C 180,E1 -24476.339,E2 -24476.339} C_VEL
LIN {X 0,Y 184.341,Z 767.235,A -85,B 0,C 180,E1 -24478.609,E2 -24478.609} C_VEL
LIN {X 0,Y 189.764,Z 756.908,A -85,B 0,C 180,E1 -24480.677,E2 -24480.677} C_VEL
LIN {X 0,Y 194.806,Z 745.294,A -85,B 0,C 180,E1 -24482.471,E2 -24482.471} C_VEL
LIN {X 0,Y 199.176,Z 732.397,A -85,B 0,C 180,E1 -24483.935,E2 -24483.935} C_VEL
LIN {X 0,Y 202.09,Z 720.863,A -85,B 0,C 180,E1 -24484.943,E2 -24484.943} C_VEL
LIN {X 0,Y 204.324,Z 708.176,A -85,B 0,C 180,E1 -24485.736,E2 -24485.736} C_VEL
LIN {X 0,Y 206.801,Z 687.22,A -85,B 0,C 180,E1 -24486.573,E2 -24486.573} C_VEL
LIN {X 0,Y 204.629,Z 681.984,A -85,B 0,C 180,E1 -24488.942,E2 -24488.942} C_VEL
LIN {X 0,Y 202.532,Z 678.371,A -85,B 0,C 180,E1 -24491.483,E2 -24491.483} C_VEL
LIN {X 0,Y 201.439,Z 676.137,A -85,B 0,C 180,E1 -24493.187,E2 -24493.187} C_VEL
LIN {X 0,Y 199.865,Z 672.877,A -85,B 0,C 180,E1 -24496.547,E2 -24496.547} C_VEL
LIN {X 0,Y 198.718,Z 672.081,A -85,B 0,C 180,E1 -24500.712,E2 -24500.712} C_VEL
LIN {X 0,Y 198.569,Z 672.74,A -85,B 0,C 180,E1 -24503.473,E2 -24503.473} C_VEL
LIN {X 0,Y 198.824,Z 674.476,A -85,B 0,C 180,E1 -24506.168,E2 -24506.168} C_VEL
LIN {X 0,Y 200.166,Z 678.667,A -85,B 0,C 180,E1 -24510.227,E2 -24510.227} C_VEL
LIN {X 0,Y 201.804,Z 683.888,A -85,B 0,C 180,E1 -24513.301,E2 -24513.301} C_VEL
LIN {X 0,Y 203.416,Z 689.15,A -85,B 0,C 180,E1 -24515.619,E2 -24515.619} C_VEL
LIN {X 0,Y 204.791,Z 694.098,A -85,B 0,C 180,E1 -24517.399,E2 -24517.399} C_VEL
LIN {X 0,Y 205.552,Z 697.44,A -85,B 0,C 180,E1 -24518.332,E2 -24518.332} C_VEL
LIN {X 0,Y 205.094,Z 704.965,A -85,B 0,C 180,E1 -24518.892,E2 -24518.892} C_VEL
LIN {X 0,Y 202.4,Z 725.112,A -85,B 0,C 180,E1 -24519.645,E2 -24519.645} C_VEL
LIN {X 0,Y 199.408,Z 738.641,A -85,B 0,C 180,E1 -24520.382,E2 -24520.382} C_VEL
LIN {X 0,Y 195.455,Z 751.328,A -85,B 0,C 180,E1 -24521.359,E2 -24521.359} C_VEL
LIN {X 0,Y 190.159,Z 764.515,A -85,B 0,C 180,E1 -24522.732,E2 -24522.732} C_VEL
LIN {X 0,Y 183.833,Z 777.251,A -85,B 0,C 180,E1 -24524.6,E2 -24524.6} C_VEL
LIN {X 0,Y 179.898,Z 784.207,A -85,B 0,C 180,E1 -24525.932,E2 -24525.932} C_VEL
LIN {X 0,Y 176.825,Z 788.622,A -85,B 0,C 180,E1 -24526.752,E2 -24526.752} C_VEL
LIN {X 0,Y 170.422,Z 795.51,A -85,B 0,C 180,E1 -24527.823,E2 -24527.823} C_VEL
LIN {X 0,Y 163.789,Z 801.757,A -85,B 0,C 180,E1 -24529.103,E2 -24529.103} C_VEL
LIN {X 0,Y 160.418,Z 805.215,A -85,B 0,C 180,E1 -24530.256,E2 -24530.256} C_VEL
LIN {X 0,Y 154.095,Z 812.214,A -85,B 0,C 180,E1 -24533.637,E2 -24533.637} C_VEL
LIN {X 0,Y 148.875,Z 817.526,A -85,B 0,C 180,E1 -24537.121,E2 -24537.121} C_VEL
LIN {X 0,Y 143.438,Z 822.701,A -85,B 0,C 180,E1 -24541.878,E2 -24541.878} C_VEL
LIN {X 0,Y 139.608,Z 825.985,A -85,B 0,C 180,E1 -24546.252,E2 -24546.252} C_VEL
LIN {X 0,Y 136.177,Z 828.637,A -85,B 0,C 180,E1 -24551.962,E2 -24551.962} C_VEL
LIN {X 0,Y 134.422,Z 829.786,A -85,B 0,C 180,E1 -24557.929,E2 -24557.929} C_VEL
LIN {X 0,Y 134.256,Z 829.439,A -85,B 0,C 180,E1 -24564.049,E2 -24564.049} C_VEL
LIN {X 0,Y 134.821,Z 827.878,A -85,B 0,C 180,E1 -24569.253,E2 -24569.253} C_VEL
LIN {X 0,Y 134.911,Z 828.156,A -85,B 0,C 180,E1 -24570,E2 -24570} C_VEL
LIN {X 0,Y 134.178,Z 829.432,A -85,B 0,C 180,E1 -24576.013,E2 -24576.013} C_VEL
LIN {X 0,Y 134.423,Z 829.049,A -85,B 0,C 180,E1 -24582.071,E2 -24582.071} C_VEL
LIN {X 0,Y 136.191,Z 827.139,A -85,B 0,C 180,E1 -24588.036,E2 -24588.036} C_VEL
LIN {X 0,Y 137.731,Z 825.572,A -85,B 0,C 180,E1 -24590.927,E2 -24590.927} C_VEL
LIN {X 0,Y 141.705,Z 821.161,A -85,B 0,C 180,E1 -24596.51,E2 -24596.51} C_VEL
LIN {X 0,Y 145.563,Z 816.633,A -85,B 0,C 180,E1 -24600.46,E2 -24600.46} C_VEL
LIN {X 0,Y 151.126,Z 809.835,A -85,B 0,C 180,E1 -24604.727,E2 -24604.727} C_VEL
LIN {X 0,Y 156.618,Z 802.478,A -85,B 0,C 180,E1 -24608.097,E2 -24608.097} C_VEL
LIN {X 0,Y 162.728,Z 793.387,A -85,B 0,C 180,E1 -24611.194,E2 -24611.194} C_VEL
LIN {X 0,Y 168.215,Z 783.959,A -85,B 0,C 180,E1 -24613.579,E2 -24613.579} C_VEL
LIN {X 0,Y 173.457,Z 773.539,A -85,B 0,C 180,E1 -24615.569,E2 -24615.569} C_VEL
LIN {X 0,Y 178.35,Z 761.943,A -85,B 0,C 180,E1 -24617.215,E2 -24617.215} C_VEL
LIN {X 0,Y 182.432,Z 749.609,A -85,B 0,C 180,E1 -24618.486,E2 -24618.486} C_VEL
LIN {X 0,Y 185.554,Z 736.896,A -85,B 0,C 180,E1 -24619.43,E2 -24619.43} C_VEL
LIN {X 0,Y 187.593,Z 724.292,A -85,B 0,C 180,E1 -24620.042,E2 -24620.042} C_VEL
LIN {X 0,Y 189.705,Z 698.297,A -85,B 0,C 180,E1 -24620.922,E2 -24620.922} C_VEL
LIN {X 0,Y 189.481,Z 685.089,A -85,B 0,C 180,E1 -24621.918,E2 -24621.918} C_VEL
LIN {X 0,Y 187.973,Z 679.605,A -85,B 0,C 180,E1 -24623.017,E2 -24623.017} C_VEL
LIN {X 0,Y 183.214,Z 670.448,A -85,B 0,C 180,E1 -24626.205,E2 -24626.205} C_VEL
LIN {X 0,Y 179.918,Z 664.711,A -85,B 0,C 180,E1 -24628.698,E2 -24628.698} C_VEL
LIN {X 0,Y 175.434,Z 657.939,A -85,B 0,C 180,E1 -24632.568,E2 -24632.568} C_VEL
LIN {X 0,Y 172.207,Z 653.447,A -85,B 0,C 180,E1 -24635.913,E2 -24635.913} C_VEL
LIN {X 0,Y 169.699,Z 649.916,A -85,B 0,C 180,E1 -24639.092,E2 -24639.092} C_VEL
LIN {X 0,Y 169.116,Z 649.037,A -85,B 0,C 180,E1 -24639.949,E2 -24639.949} C_VEL
LIN {X 0,Y 166.661,Z 646.072,A -85,B 0,C 180,E1 -24644.321,E2 -24644.321} C_VEL
LIN {X 0,Y 165.915,Z 644.126,A -85,B 0,C 180,E1 -24646.418,E2 -24646.418} C_VEL
LIN {X 0,Y 164.445,Z 643.141,A -85,B 0,C 180,E1 -24652.634,E2 -24652.634} C_VEL
LIN {X 0,Y 164.836,Z 643.138,A -85,B 0,C 180,E1 -24658.778,E2 -24658.778} C_VEL
LIN {X 0,Y 166.128,Z 644.083,A -85,B 0,C 180,E1 -24663.015,E2 -24663.015} C_VEL
LIN {X 0,Y 167.631,Z 647.204,A -85,B 0,C 180,E1 -24666.545,E2 -24666.545} C_VEL
LIN {X 0,Y 169.522,Z 649.276,A -85,B 0,C 180,E1 -24669.546,E2 -24669.546} C_VEL
LIN {X 0,Y 171.906,Z 653.017,A -85,B 0,C 180,E1 -24672.694,E2 -24672.694} C_VEL
LIN {X 0,Y 173.041,Z 654.477,A -85,B 0,C 180,E1 -24673.954,E2 -24673.954} C_VEL
LIN {X 0,Y 176.306,Z 659.229,A -85,B 0,C 180,E1 -24677.195,E2 -24677.195} C_VEL
LIN {X 0,Y 179.195,Z 663.677,A -85,B 0,C 180,E1 -24679.68,E2 -24679.68} C_VEL
LIN {X 0,Y 183.031,Z 669.8,A -85,B 0,C 180,E1 -24682.58,E2 -24682.58} C_VEL
LIN {X 0,Y 188.092,Z 678.66,A -85,B 0,C 180,E1 -24685.922,E2 -24685.922} C_VEL
LIN {X 0,Y 190.991,Z 684.337,A -85,B 0,C 180,E1 -24687.664,E2 -24687.664} C_VEL
LIN {X 0,Y 189.206,Z 707.81,A -85,B 0,C 180,E1 -24688.588,E2 -24688.588} C_VEL
LIN {X 0,Y 187.136,Z 720.777,A -85,B 0,C 180,E1 -24689.416,E2 -24689.416} C_VEL
LIN {X 0,Y 184.157,Z 733.347,A -85,B 0,C 180,E1 -24690.567,E2 -24690.567} C_VEL
LIN {X 0,Y 180.45,Z 745.193,A -85,B 0,C 180,E1 -24692.105,E2 -24692.105} C_VEL
LIN {X 0,Y 175.973,Z 756.399,A -85,B 0,C 180,E1 -24693.996,E2 -24693.996} C_VEL
LIN {X 0,Y 171.499,Z 765.585,A -85,B 0,C 180,E1 -24695.969,E2 -24695.969} C_VEL
LIN {X 0,Y 166.217,Z 774.814,A -85,B 0,C 180,E1 -24698.538,E2 -24698.538} C_VEL
LIN {X 0,Y 160.35,Z 783.685,A -85,B 0,C 180,E1 -24701.835,E2 -24701.835} C_VEL
LIN {X 0,Y 154.974,Z 790.72,A -85,B 0,C 180,E1 -24705.34,E2 -24705.34} C_VEL
LIN {X 0,Y 150.122,Z 796.244,A -85,B 0,C 180,E1 -24709.05,E2 -24709.05} C_VEL
LIN {X 0,Y 145.867,Z 800.503,A -85,B 0,C 180,E1 -24712.969,E2 -24712.969} C_VEL
LIN {X 0,Y 142.223,Z 803.671,A -85,B 0,C 180,E1 -24717.147,E2 -24717.147} C_VEL
LIN {X 0,Y 140.255,Z 805.154,A -85,B 0,C 180,E1 -24719.929,E2 -24719.929} C_VEL
LIN {X 0,Y 138.518,Z 806.235,A -85,B 0,C 180,E1 -24722.831,E2 -24722.831} C_VEL
LIN {X 0,Y 136.05,Z 807.099,A -85,B 0,C 180,E1 -24728.802,E2 -24728.802} C_VEL
LIN {X 0,Y 135.194,Z 806.942,A -85,B 0,C 180,E1 -24731.826,E2 -24731.826} C_VEL
LIN {X 0,Y 134.648,Z 806.335,A -85,B 0,C 180,E1 -24734.872,E2 -24734.872} C_VEL
LIN {X 0,Y 134.415,Z 805.331,A -85,B 0,C 180,E1 -24737.928,E2 -24737.928} C_VEL
LIN {X 0,Y 134.597,Z 802.874,A -85,B 0,C 180,E1 -24742.79,E2 -24742.79} C_VEL
LIN {X 0,Y 135.305,Z 799.785,A -85,B 0,C 180,E1 -24747.023,E2 -24747.023} C_VEL
LIN {X 0,Y 136.564,Z 795.463,A -85,B 0,C 180,E1 -24751.474,E2 -24751.474} C_VEL
LIN {X 0,Y 138.391,Z 789.963,A -85,B 0,C 180,E1 -24755.829,E2 -24755.829} C_VEL
LIN {X 0,Y 140.791,Z 783.09,A -85,B 0,C 180,E1 -24760.062,E2 -24760.062} C_VEL
LIN {X 0,Y 143.845,Z 774.46,A -85,B 0,C 180,E1 -24764.14,E2 -24764.14} C_VEL
LIN {X 0,Y 146.901,Z 765.614,A -85,B 0,C 180,E1 -24767.398,E2 -24767.398} C_VEL
LIN {X 0,Y 144.342,Z 763.078,A -85,B 0,C 180,E1 -24768.956,E2 -24768.956} C_VEL
LIN {X 0,Y 141.949,Z 771.823,A -85,B 0,C 180,E1 -24772.059,E2 -24772.059} C_VEL
LIN {X 0,Y 139.336,Z 780.812,A -85,B 0,C 180,E1 -24776.065,E2 -24776.065} C_VEL
LIN {X 0,Y 137.099,Z 789.162,A -85,B 0,C 180,E1 -24780.838,E2 -24780.838} C_VEL
LIN {X 0,Y 135.498,Z 795.614,A -85,B 0,C 180,E1 -24785.666,E2 -24785.666} C_VEL
LIN {X 0,Y 134.517,Z 800.812,A -85,B 0,C 180,E1 -24790.773,E2 -24790.773} C_VEL
LIN {X 0,Y 134.243,Z 804.013,A -85,B 0,C 180,E1 -24794.969,E2 -24794.969} C_VEL
LIN {X 0,Y 134.556,Z 806.412,A -85,B 0,C 180,E1 -24799.24,E2 -24799.24} C_VEL
LIN {X 0,Y 136.095,Z 808.436,A -85,B 0,C 180,E1 -24805.386,E2 -24805.386} C_VEL
LIN {X 0,Y 138.075,Z 808.838,A -85,B 0,C 180,E1 -24809.914,E2 -24809.914} C_VEL
LIN {X 0,Y 140.613,Z 808.343,A -85,B 0,C 180,E1 -24814.11,E2 -24814.11} C_VEL
LIN {X 0,Y 143.84,Z 806.976,A -85,B 0,C 180,E1 -24818.173,E2 -24818.173} C_VEL
LIN {X 0,Y 147.711,Z 804.678,A -85,B 0,C 180,E1 -24822.095,E2 -24822.095} C_VEL
LIN {X 0,Y 153.517,Z 800.376,A -85,B 0,C 180,E1 -24826.768,E2 -24826.768} C_VEL
LIN {X 0,Y 159.156,Z 795.336,A -85,B 0,C 180,E1 -24830.468,E2 -24830.468} C_VEL
LIN {X 0,Y 165.434,Z 788.741,A -85,B 0,C 180,E1 -24833.934,E2 -24833.934} C_VEL
LIN {X 0,Y 171.353,Z 781.599,A -85,B 0,C 180,E1 -24836.727,E2 -24836.727} C_VEL
LIN {X 0,Y 177.487,Z 773.045,A -85,B 0,C 180,E1 -24839.31,E2 -24839.31} C_VEL
LIN {X 0,Y 183.649,Z 762.82,A -85,B 0,C 180,E1 -24841.634,E2 -24841.634} C_VEL
LIN {X 0,Y 189.244,Z 751.656,A -85,B 0,C 180,E1 -24843.546,E2 -24843.546} C_VEL
LIN {X 0,Y 193.548,Z 741.075,A -85,B 0,C 180,E1 -24844.947,E2 -24844.947} C_VEL
LIN {X 0,Y 197.625,Z 728.18,A -85,B 0,C 180,E1 -24846.257,E2 -24846.257} C_VEL
LIN {X 0,Y 200.64,Z 715.035,A -85,B 0,C 180,E1 -24847.235,E2 -24847.235} C_VEL
LIN {X 0,Y 202.552,Z 701.842,A -85,B 0,C 180,E1 -24847.889,E2 -24847.889} C_VEL
LIN {X 0,Y 203.817,Z 691.202,A -85,B 0,C 180,E1 -24848.324,E2 -24848.324} C_VEL
LIN {X 0,Y 202.667,Z 688.209,A -85,B 0,C 180,E1 -24849.721,E2 -24849.721} C_VEL
LIN {X 0,Y 199.911,Z 682.812,A -85,B 0,C 180,E1 -24853.728,E2 -24853.728} C_VEL
LIN {X 0,Y 198.49,Z 679.781,A -85,B 0,C 180,E1 -24857.065,E2 -24857.065} C_VEL
LIN {X 0,Y 197.562,Z 679.088,A -85,B 0,C 180,E1 -24860.839,E2 -24860.839} C_VEL
LIN {X 0,Y 197.427,Z 679.882,A -85,B 0,C 180,E1 -24863.617,E2 -24863.617} C_VEL
LIN {X 0,Y 197.653,Z 681.706,A -85,B 0,C 180,E1 -24866.182,E2 -24866.182} C_VEL
LIN {X 0,Y 198.631,Z 685.107,A -85,B 0,C 180,E1 -24869.473,E2 -24869.473} C_VEL
LIN {X 0,Y 199.974,Z 689.927,A -85,B 0,C 180,E1 -24872.364,E2 -24872.364} C_VEL
LIN {X 0,Y 201.255,Z 694.771,A -85,B 0,C 180,E1 -24874.553,E2 -24874.553} C_VEL
LIN {X 0,Y 202.388,Z 699.203,A -85,B 0,C 180,E1 -24876.181,E2 -24876.181} C_VEL
LIN {X 0,Y 202.746,Z 700.83,A -85,B 0,C 180,E1 -24876.697,E2 -24876.697} C_VEL
LIN {X 0,Y 202.333,Z 706.086,A -85,B 0,C 180,E1 -24877.079,E2 -24877.079} C_VEL
LIN {X 0,Y 199.52,Z 725.501,A -85,B 0,C 180,E1 -24877.799,E2 -24877.799} C_VEL
LIN {X 0,Y 196.446,Z 738.514,A -85,B 0,C 180,E1 -24878.503,E2 -24878.503} C_VEL
LIN {X 0,Y 192.312,Z 751.248,A -85,B 0,C 180,E1 -24879.467,E2 -24879.467} C_VEL
LIN {X 0,Y 187.524,Z 762.825,A -85,B 0,C 180,E1 -24880.632,E2 -24880.632} C_VEL
LIN {X 0,Y 181.569,Z 774.598,A -85,B 0,C 180,E1 -24882.247,E2 -24882.247} C_VEL
LIN {X 0,Y 175.36,Z 785.03,A -85,B 0,C 180,E1 -24884.198,E2 -24884.198} C_VEL
LIN {X 0,Y 168.671,Z 794.677,A -85,B 0,C 180,E1 -24886.569,E2 -24886.569} C_VEL
LIN {X 0,Y 162.089,Z 803.181,A -85,B 0,C 180,E1 -24889.431,E2 -24889.431} C_VEL
LIN {X 0,Y 160.418,Z 805.215,A -85,B 0,C 180,E1 -24890.256,E2 -24890.256} C_VEL
LIN {X 0,Y 157.011,Z 808.536,A -85,B 0,C 180,E1 -24891.529,E2 -24891.529} C_VEL
LIN {X 0,Y 150.139,Z 813.464,A -85,B 0,C 180,E1 -24893.472,E2 -24893.472} C_VEL
LIN {X 0,Y 143.423,Z 817.721,A -85,B 0,C 180,E1 -24895.764,E2 -24895.764} C_VEL
LIN {X 0,Y 140.343,Z 819.929,A -85,B 0,C 180,E1 -24897.577,E2 -24897.577} C_VEL
LIN {X 0,Y 135.517,Z 823.909,A -85,B 0,C 180,E1 -24902.178,E2 -24902.178} C_VEL
LIN {X 0,Y 131.097,Z 827.139,A -85,B 0,C 180,E1 -24907.96,E2 -24907.96} C_VEL
LIN {X 0,Y 128.232,Z 828.812,A -85,B 0,C 180,E1 -24914.096,E2 -24914.096} C_VEL
LIN {X 0,Y 127.121,Z 829.055,A -85,B 0,C 180,E1 -24920.453,E2 -24920.453} C_VEL
LIN {X 0,Y 127.206,Z 828.569,A -85,B 0,C 180,E1 -24923.978,E2 -24923.978} C_VEL
LIN {X 0,Y 127.735,Z 827.076,A -85,B 0,C 180,E1 -24929.015,E2 -24929.015} C_VEL
LIN {X 0,Y 127.846,Z 827.453,A -85,B 0,C 180,E1 -24930,E2 -24930} C_VEL
LIN {X 0,Y 127.077,Z 828.779,A -85,B 0,C 180,E1 -24936.35,E2 -24936.35} C_VEL
LIN {X 0,Y 127.054,Z 828.842,A -85,B 0,C 180,E1 -24939.552,E2 -24939.552} C_VEL
LIN {X 0,Y 128.243,Z 827.748,A -85,B 0,C 180,E1 -24945.903,E2 -24945.903} C_VEL
LIN {X 0,Y 129.427,Z 826.634,A -85,B 0,C 180,E1 -24949.014,E2 -24949.014} C_VEL
LIN {X 0,Y 131.084,Z 825.125,A -85,B 0,C 180,E1 -24952.042,E2 -24952.042} C_VEL
LIN {X 0,Y 134.172,Z 822.05,A -85,B 0,C 180,E1 -24956.438,E2 -24956.438} C_VEL
LIN {X 0,Y 137.992,Z 817.953,A -85,B 0,C 180,E1 -24960.617,E2 -24960.617} C_VEL
LIN {X 0,Y 143.584,Z 811.714,A -85,B 0,C 180,E1 -24965.107,E2 -24965.107} C_VEL
